LIN {X 0,Y 488.763,Z 747.858,A -85,B 0,C 180,E1 22935.063,E2 22935.063} C_VEL
LIN {X 0,Y 489.433,Z 736.714,A -85,B 0,C 180,E1 22932.524,E2 22932.524} C_VEL
LIN {X 0,Y 490.367,Z 723.912,A -85,B 0,C 180,E1 22930.092,E2 22930.092} C_VEL
LIN {X 0,Y 491.563,Z 709.449,A -85,B 0,C 180,E1 22927.769,E2 22927.769} C_VEL
LIN {X 0,Y 493.023,Z 693.233,A -85,B 0,C 180,E1 22925.561,E2 22925.561} C_VEL
LIN {X 0,Y 494.639,Z 676.036,A -85,B 0,C 180,E1 22923.569,E2 22923.569} C_VEL
LIN {X 0,Y 496.38,Z 657.448,A -85,B 0,C 180,E1 22921.747,E2 22921.747} C_VEL
LIN {X 0,Y 498.101,Z 638.983,A -85,B 0,C 180,E1 22920.21,E2 22920.21} C_VEL
LIN {X 0,Y 499.849,Z 618.816,A -85,B 0,C 180,E1 22918.796,E2 22918.796} C_VEL
LIN {X 0,Y 501.367,Z 599.666,A -85,B 0,C 180,E1 22917.692,E2 22917.692} C_VEL
LIN {X 0,Y 502.665,Z 578.619,A -85,B 0,C 180,E1 22916.736,E2 22916.736} C_VEL
LIN {X 0,Y 503.879,Z 555.736,A -85,B 0,C 180,E1 22915.926,E2 22915.926} C_VEL
LIN {X 0,Y 504.882,Z 532.422,A -85,B 0,C 180,E1 22915.329,E2 22915.329} C_VEL
LIN {X 0,Y 505.632,Z 495.194,A -85,B 0,C 180,E1 22914.703,E2 22914.703} C_VEL
LIN {X 0,Y 506.044,Z 485.944,A -85,B 0,C 180,E1 22914.556,E2 22914.556} C_VEL
LIN {X 0,Y 510.084,Z 468.745,A -85,B 0,C 180,E1 22913.911,E2 22913.911} C_VEL
LIN {X 0,Y 515.233,Z 449.255,A -85,B 0,C 180,E1 22913.225,E2 22913.225} C_VEL
LIN {X 0,Y 520.98,Z 432.729,A -85,B 0,C 180,E1 22912.735,E2 22912.735} C_VEL
LIN {X 0,Y 525.125,Z 418.193,A -85,B 0,C 180,E1 22912.255,E2 22912.255} C_VEL
LIN {X 0,Y 532.74,Z 398.375,A -85,B 0,C 180,E1 22911.731,E2 22911.731} C_VEL
LIN {X 0,Y 544.808,Z 371.898,A -85,B 0,C 180,E1 22911.19,E2 22911.19} C_VEL
LIN {X 0,Y 552.914,Z 353.703,A -85,B 0,C 180,E1 22910.934,E2 22910.934} C_VEL
LIN {X 0,Y 556.995,Z 340.142,A -85,B 0,C 180,E1 22910.569,E2 22910.569} C_VEL
LIN {X 0,Y 565.45,Z 316.224,A -85,B 0,C 180,E1 22910.17,E2 22910.17} C_VEL
LIN {X 0,Y 574.832,Z 288.327,A -85,B 0,C 180,E1 22909.898,E2 22909.898} C_VEL
LIN {X 0,Y 577.335,Z 280.017,A -85,B 0,C 180,E1 22909.834,E2 22909.834} C_VEL
LIN {X 0,Y 575.602,Z 280.443,A -85,B 0,C 180,E1 22909.221,E2 22909.221} C_VEL
LIN {X 0,Y 572.536,Z 280.47,A -85,B 0,C 180,E1 22908.671,E2 22908.671} C_VEL
LIN {X 0,Y 567.829,Z 279.596,A -85,B 0,C 180,E1 22908.145,E2 22908.145} C_VEL
LIN {X 0,Y 556.51,Z 275.352,A -85,B 0,C 180,E1 22907.141,E2 22907.141} C_VEL
LIN {X 0,Y 546.549,Z 269.641,A -85,B 0,C 180,E1 22906.119,E2 22906.119} C_VEL
LIN {X 0,Y 532.658,Z 258.791,A -85,B 0,C 180,E1 22904.44,E2 22904.44} C_VEL
LIN {X 0,Y 524.421,Z 249.344,A -85,B 0,C 180,E1 22903.193,E2 22903.193} C_VEL
LIN {X 0,Y 518.357,Z 238.972,A -85,B 0,C 180,E1 22902.015,E2 22902.015} C_VEL
LIN {X 0,Y 507.707,Z 216,A -85,B 0,C 180,E1 22899.467,E2 22899.467} C_VEL
LIN {X 0,Y 499.256,Z 199.711,A -85,B 0,C 180,E1 22897.359,E2 22897.359} C_VEL
LIN {X 0,Y 493.765,Z 190.209,A -85,B 0,C 180,E1 22895.961,E2 22895.961} C_VEL
LIN {X 0,Y 491.774,Z 186.487,A -85,B 0,C 180,E1 22895.412,E2 22895.412} C_VEL
LIN {X 0,Y 489.247,Z 182.669,A -85,B 0,C 180,E1 22894.759,E2 22894.759} C_VEL
LIN {X 0,Y 488.789,Z 180.844,A -85,B 0,C 180,E1 22894.515,E2 22894.515} C_VEL
LIN {X 0,Y 488.82,Z 181.07,A -85,B 0,C 180,E1 22894.37,E2 22894.37} C_VEL
LIN {X 0,Y 493.804,Z 196.293,A -85,B 0,C 180,E1 22893.002,E2 22893.002} C_VEL
LIN {X 0,Y 494.732,Z 233.032,A -85,B 0,C 180,E1 22890.281,E2 22890.281} C_VEL
LIN {X 0,Y 495.182,Z 268.429,A -85,B 0,C 180,E1 22887.476,E2 22887.476} C_VEL
LIN {X 0,Y 495.112,Z 303.332,A -85,B 0,C 180,E1 22884.582,E2 22884.582} C_VEL
LIN {X 0,Y 494.717,Z 328.2,A -85,B 0,C 180,E1 22882.456,E2 22882.456} C_VEL
LIN {X 0,Y 494.316,Z 330.636,A -85,B 0,C 180,E1 22882.319,E2 22882.319} C_VEL
LIN {X 0,Y 492.834,Z 451.64,A -85,B 0,C 180,E1 22880.353,E2 22880.353} C_VEL
LIN {X 0,Y 492.642,Z 497.502,A -85,B 0,C 180,E1 22879.623,E2 22879.623} C_VEL
LIN {X 0,Y 492.552,Z 514.82,A -85,B 0,C 180,E1 22879.126,E2 22879.126} C_VEL
LIN {X 0,Y 492.299,Z 531.833,A -85,B 0,C 180,E1 22878.41,E2 22878.41} C_VEL
LIN {X 0,Y 491.931,Z 547.816,A -85,B 0,C 180,E1 22877.506,E2 22877.506} C_VEL
LIN {X 0,Y 491.461,Z 562.541,A -85,B 0,C 180,E1 22876.426,E2 22876.426} C_VEL
LIN {X 0,Y 490.921,Z 576.831,A -85,B 0,C 180,E1 22875.111,E2 22875.111} C_VEL
LIN {X 0,Y 490.398,Z 589.354,A -85,B 0,C 180,E1 22873.68,E2 22873.68} C_VEL
LIN {X 0,Y 489.896,Z 600.231,A -85,B 0,C 180,E1 22872.135,E2 22872.135} C_VEL
LIN {X 0,Y 489.44,Z 610.273,A -85,B 0,C 180,E1 22870.356,E2 22870.356} C_VEL
LIN {X 0,Y 489.118,Z 618.168,A -85,B 0,C 180,E1 22868.582,E2 22868.582} C_VEL
LIN {X 0,Y 488.849,Z 624.536,A -85,B 0,C 180,E1 22866.695,E2 22866.695} C_VEL
LIN {X 0,Y 488.668,Z 629.357,A -85,B 0,C 180,E1 22864.694,E2 22864.694} C_VEL
LIN {X 0,Y 488.565,Z 632.392,A -85,B 0,C 180,E1 22862.698,E2 22862.698} C_VEL
LIN {X 0,Y 488.509,Z 633.701,A -85,B 0,C 180,E1 22860.703,E2 22860.703} C_VEL
LIN {X 0,Y 488.489,Z 633.33,A -85,B 0,C 180,E1 22858.709,E2 22858.709} C_VEL
LIN {X 0,Y 488.513,Z 631.151,A -85,B 0,C 180,E1 22856.597,E2 22856.597} C_VEL
LIN {X 0,Y 488.59,Z 627.335,A -85,B 0,C 180,E1 22854.598,E2 22854.598} C_VEL
LIN {X 0,Y 488.748,Z 621.608,A -85,B 0,C 180,E1 22852.595,E2 22852.595} C_VEL
LIN {X 0,Y 489.001,Z 614.344,A -85,B 0,C 180,E1 22850.704,E2 22850.704} C_VEL
LIN {X 0,Y 489.348,Z 605.609,A -85,B 0,C 180,E1 22848.926,E2 22848.926} C_VEL
LIN {X 0,Y 489.79,Z 595.341,A -85,B 0,C 180,E1 22847.263,E2 22847.263} C_VEL
LIN {X 0,Y 490.348,Z 583.074,A -85,B 0,C 180,E1 22845.655,E2 22845.655} C_VEL
LIN {X 0,Y 490.92,Z 570.214,A -85,B 0,C 180,E1 22844.283,E2 22844.283} C_VEL
LIN {X 0,Y 491.478,Z 556.401,A -85,B 0,C 180,E1 22843.087,E2 22843.087} C_VEL
LIN {X 0,Y 492.034,Z 540.803,A -85,B 0,C 180,E1 22842.008,E2 22842.008} C_VEL
LIN {X 0,Y 492.492,Z 524.476,A -85,B 0,C 180,E1 22841.129,E2 22841.129} C_VEL
LIN {X 0,Y 492.864,Z 507.517,A -85,B 0,C 180,E1 22840.456,E2 22840.456} C_VEL
LIN {X 0,Y 493.062,Z 489.747,A -85,B 0,C 180,E1 22839.985,E2 22839.985} C_VEL
LIN {X 0,Y 494.563,Z 326.51,A -85,B 0,C 180,E1 22837.4,E2 22837.4} C_VEL
LIN {X 0,Y 493.777,Z 321.369,A -85,B 0,C 180,E1 22837.246,E2 22837.246} C_VEL
LIN {X 0,Y 494.7,Z 284.617,A -85,B 0,C 180,E1 22833.817,E2 22833.817} C_VEL
LIN {X 0,Y 495.483,Z 247.552,A -85,B 0,C 180,E1 22830.369,E2 22830.369} C_VEL
LIN {X 0,Y 495.924,Z 219.277,A -85,B 0,C 180,E1 22827.745,E2 22827.745} C_VEL
LIN {X 0,Y 496.216,Z 218.46,A -85,B 0,C 180,E1 22827.507,E2 22827.507} C_VEL
LIN {X 0,Y 497.105,Z 219.551,A -85,B 0,C 180,E1 22827.105,E2 22827.105} C_VEL
LIN {X 0,Y 498.497,Z 223.242,A -85,B 0,C 180,E1 22826.646,E2 22826.646} C_VEL
LIN {X 0,Y 500.085,Z 229.6,A -85,B 0,C 180,E1 22826.249,E2 22826.249} C_VEL
LIN {X 0,Y 501.866,Z 239.61,A -85,B 0,C 180,E1 22825.842,E2 22825.842} C_VEL
LIN {X 0,Y 502.271,Z 247.308,A -85,B 0,C 180,E1 22825.659,E2 22825.659} C_VEL
LIN {X 0,Y 498.516,Z 445.436,A -85,B 0,C 180,E1 22822.414,E2 22822.414} C_VEL
LIN {X 0,Y 497.797,Z 472.996,A -85,B 0,C 180,E1 22821.899,E2 22821.899} C_VEL
LIN {X 0,Y 496.838,Z 494.838,A -85,B 0,C 180,E1 22821.269,E2 22821.269} C_VEL
LIN {X 0,Y 495.591,Z 515.448,A -85,B 0,C 180,E1 22820.462,E2 22820.462} C_VEL
LIN {X 0,Y 494.06,Z 535.344,A -85,B 0,C 180,E1 22819.458,E2 22819.458} C_VEL
LIN {X 0,Y 492.584,Z 552.464,A -85,B 0,C 180,E1 22818.413,E2 22818.413} C_VEL
LIN {X 0,Y 490.672,Z 572.409,A -85,B 0,C 180,E1 22816.949,E2 22816.949} C_VEL
LIN {X 0,Y 489.001,Z 588.827,A -85,B 0,C 180,E1 22815.529,E2 22815.529} C_VEL
LIN {X 0,Y 487.387,Z 604.827,A -85,B 0,C 180,E1 22813.939,E2 22813.939} C_VEL
LIN {X 0,Y 485.617,Z 622.035,A -85,B 0,C 180,E1 22811.938,E2 22811.938} C_VEL
LIN {X 0,Y 484.269,Z 635.641,A -85,B 0,C 180,E1 22810.104,E2 22810.104} C_VEL
LIN {X 0,Y 482.989,Z 649.658,A -85,B 0,C 180,E1 22807.933,E2 22807.933} C_VEL
LIN {X 0,Y 482.001,Z 661.364,A -85,B 0,C 180,E1 22805.797,E2 22805.797} C_VEL
LIN {X 0,Y 481.217,Z 672.009,A -85,B 0,C 180,E1 22803.552,E2 22803.552} C_VEL
LIN {X 0,Y 480.597,Z 682.358,A -85,B 0,C 180,E1 22800.922,E2 22800.922} C_VEL
LIN {X 0,Y 480.254,Z 689.801,A -85,B 0,C 180,E1 22798.61,E2 22798.61} C_VEL
LIN {X 0,Y 480.033,Z 696.665,A -85,B 0,C 180,E1 22795.939,E2 22795.939} C_VEL
LIN {X 0,Y 479.947,Z 701.157,A -85,B 0,C 180,E1 22793.559,E2 22793.559} C_VEL
LIN {X 0,Y 479.92,Z 704.361,A -85,B 0,C 180,E1 22791.127,E2 22791.127} C_VEL
LIN {X 0,Y 479.9,Z 706.187,A -85,B 0,C 180,E1 22788.463,E2 22788.463} C_VEL
LIN {X 0,Y 479.914,Z 706.33,A -85,B 0,C 180,E1 22786.087,E2 22786.087} C_VEL
LIN {X 0,Y 479.917,Z 705.127,A -85,B 0,C 180,E1 22783.617,E2 22783.617} C_VEL
LIN {X 0,Y 479.936,Z 702.064,A -85,B 0,C 180,E1 22780.929,E2 22780.929} C_VEL
LIN {X 0,Y 480,Z 697.765,A -85,B 0,C 180,E1 22778.505,E2 22778.505} C_VEL
LIN {X 0,Y 480.186,Z 691.783,A -85,B 0,C 180,E1 22775.976,E2 22775.976} C_VEL
LIN {X 0,Y 480.518,Z 683.988,A -85,B 0,C 180,E1 22773.46,E2 22773.46} C_VEL
LIN {X 0,Y 481.065,Z 674.571,A -85,B 0,C 180,E1 22770.953,E2 22770.953} C_VEL
LIN {X 0,Y 481.862,Z 663.093,A -85,B 0,C 180,E1 22768.454,E2 22768.454} C_VEL
LIN {X 0,Y 482.743,Z 652.276,A -85,B 0,C 180,E1 22766.438,E2 22766.438} C_VEL
LIN {X 0,Y 484.023,Z 638.341,A -85,B 0,C 180,E1 22764.191,E2 22764.191} C_VEL
LIN {X 0,Y 485.448,Z 623.716,A -85,B 0,C 180,E1 22762.187,E2 22762.187} C_VEL
LIN {X 0,Y 487.068,Z 608.002,A -85,B 0,C 180,E1 22760.309,E2 22760.309} C_VEL
LIN {X 0,Y 488.817,Z 590.709,A -85,B 0,C 180,E1 22758.556,E2 22758.556} C_VEL
LIN {X 0,Y 490.405,Z 574.812,A -85,B 0,C 180,E1 22757.16,E2 22757.16} C_VEL
LIN {X 0,Y 492.33,Z 555.785,A -85,B 0,C 180,E1 22755.715,E2 22755.715} C_VEL
LIN {X 0,Y 493.921,Z 537.357,A -85,B 0,C 180,E1 22754.562,E2 22754.562} C_VEL
LIN {X 0,Y 495.381,Z 518.625,A -85,B 0,C 180,E1 22753.586,E2 22753.586} C_VEL
LIN {X 0,Y 496.824,Z 496.661,A -85,B 0,C 180,E1 22752.691,E2 22752.691} C_VEL
LIN {X 0,Y 497.85,Z 474.503,A -85,B 0,C 180,E1 22752.025,E2 22752.025} C_VEL
LIN {X 0,Y 498.582,Z 449.883,A -85,B 0,C 180,E1 22751.541,E2 22751.541} C_VEL
LIN {X 0,Y 502.344,Z 259.982,A -85,B 0,C 180,E1 22748.409,E2 22748.409} C_VEL
LIN {X 0,Y 503.199,Z 216.754,A -85,B 0,C 180,E1 22747.677,E2 22747.677} C_VEL
LIN {X 0,Y 492.328,Z 199.865,A -85,B 0,C 180,E1 22746.266,E2 22746.266} C_VEL
LIN {X 0,Y 486.193,Z 190.932,A -85,B 0,C 180,E1 22745.443,E2 22745.443} C_VEL
LIN {X 0,Y 483.497,Z 186.812,A -85,B 0,C 180,E1 22745.069,E2 22745.069} C_VEL
LIN {X 0,Y 481.403,Z 183.82,A -85,B 0,C 180,E1 22744.779,E2 22744.779} C_VEL
LIN {X 0,Y 480.893,Z 181.877,A -85,B 0,C 180,E1 22744.631,E2 22744.631} C_VEL
LIN {X 0,Y 480.883,Z 181.825,A -85,B 0,C 180,E1 22741.023,E2 22741.023} C_VEL
LIN {X 0,Y 480.846,Z 181.833,A -85,B 0,C 180,E1 22737.556,E2 22737.556} C_VEL
LIN {X 0,Y 480.828,Z 181.84,A -85,B 0,C 180,E1 22733.951,E2 22733.951} C_VEL
LIN {X 0,Y 480.866,Z 181.837,A -85,B 0,C 180,E1 22730.482,E2 22730.482} C_VEL
LIN {X 0,Y 480.892,Z 181.835,A -85,B 0,C 180,E1 22727.002,E2 22727.002} C_VEL
LIN {X 0,Y 480.881,Z 181.834,A -85,B 0,C 180,E1 22723.326,E2 22723.326} C_VEL
LIN {X 0,Y 480.865,Z 181.831,A -85,B 0,C 180,E1 22719.669,E2 22719.669} C_VEL
LIN {X 0,Y 480.862,Z 181.825,A -85,B 0,C 180,E1 22716.195,E2 22716.195} C_VEL
LIN {X 0,Y 480.873,Z 181.823,A -85,B 0,C 180,E1 22712.584,E2 22712.584} C_VEL
LIN {X 0,Y 480.896,Z 181.83,A -85,B 0,C 180,E1 22708.977,E2 22708.977} C_VEL
LIN {X 0,Y 480.889,Z 181.836,A -85,B 0,C 180,E1 22705.361,E2 22705.361} C_VEL
LIN {X 0,Y 480.89,Z 181.825,A -85,B 0,C 180,E1 22701.722,E2 22701.722} C_VEL
LIN {X 0,Y 480.889,Z 181.821,A -85,B 0,C 180,E1 22698.16,E2 22698.16} C_VEL
LIN {X 0,Y 480.888,Z 181.828,A -85,B 0,C 180,E1 22694.572,E2 22694.572} C_VEL
LIN {X 0,Y 480.871,Z 181.839,A -85,B 0,C 180,E1 22690.907,E2 22690.907} C_VEL
LIN {X 0,Y 480.871,Z 181.831,A -85,B 0,C 180,E1 22687.338,E2 22687.338} C_VEL
LIN {X 0,Y 480.88,Z 181.822,A -85,B 0,C 180,E1 22683.696,E2 22683.696} C_VEL
LIN {X 0,Y 480.89,Z 181.823,A -85,B 0,C 180,E1 22680.12,E2 22680.12} C_VEL
LIN {X 0,Y 480.882,Z 181.829,A -85,B 0,C 180,E1 22676.544,E2 22676.544} C_VEL
LIN {X 0,Y 480.834,Z 181.84,A -85,B 0,C 180,E1 22673.073,E2 22673.073} C_VEL
LIN {X 0,Y 480.843,Z 181.839,A -85,B 0,C 180,E1 22669.457,E2 22669.457} C_VEL
LIN {X 0,Y 480.865,Z 181.836,A -85,B 0,C 180,E1 22665.797,E2 22665.797} C_VEL
LIN {X 0,Y 480.887,Z 181.829,A -85,B 0,C 180,E1 22662.204,E2 22662.204} C_VEL
LIN {X 0,Y 480.875,Z 181.824,A -85,B 0,C 180,E1 22658.662,E2 22658.662} C_VEL
LIN {X 0,Y 480.844,Z 181.835,A -85,B 0,C 180,E1 22655.164,E2 22655.164} C_VEL
LIN {X 0,Y 480.863,Z 181.881,A -85,B 0,C 180,E1 22653.845,E2 22653.845} C_VEL
LIN {X 0,Y 481.911,Z 184.96,A -85,B 0,C 180,E1 22653.375,E2 22653.375} C_VEL
LIN {X 0,Y 483.361,Z 187.323,A -85,B 0,C 180,E1 22652.93,E2 22652.93} C_VEL
LIN {X 0,Y 490.426,Z 201.495,A -85,B 0,C 180,E1 22650.572,E2 22650.572} C_VEL
LIN {X 0,Y 498.189,Z 217.501,A -85,B 0,C 180,E1 22648.098,E2 22648.098} C_VEL
LIN {X 0,Y 504.131,Z 230.513,A -85,B 0,C 180,E1 22646.236,E2 22646.236} C_VEL
LIN {X 0,Y 501.407,Z 270.851,A -85,B 0,C 180,E1 22642.971,E2 22642.971} C_VEL
LIN {X 0,Y 500.283,Z 297.085,A -85,B 0,C 180,E1 22640.836,E2 22640.836} C_VEL
LIN {X 0,Y 501.428,Z 313.16,A -85,B 0,C 180,E1 22639.38,E2 22639.38} C_VEL
LIN {X 0,Y 504.425,Z 327.463,A -85,B 0,C 180,E1 22637.935,E2 22637.935} C_VEL
LIN {X 0,Y 508.961,Z 339.677,A -85,B 0,C 180,E1 22636.562,E2 22636.562} C_VEL
LIN {X 0,Y 514.631,Z 349.651,A -85,B 0,C 180,E1 22635.307,E2 22635.307} C_VEL
LIN {X 0,Y 522.401,Z 359.052,A -85,B 0,C 180,E1 22633.975,E2 22633.975} C_VEL
LIN {X 0,Y 531.862,Z 366.96,A -85,B 0,C 180,E1 22632.689,E2 22632.689} C_VEL
LIN {X 0,Y 542.304,Z 372.999,A -85,B 0,C 180,E1 22631.535,E2 22631.535} C_VEL
LIN {X 0,Y 553.572,Z 377.39,A -85,B 0,C 180,E1 22630.5,E2 22630.5} C_VEL
LIN {X 0,Y 558.618,Z 378.484,A -85,B 0,C 180,E1 22629.998,E2 22629.998} C_VEL
LIN {X 0,Y 562.474,Z 378.433,A -85,B 0,C 180,E1 22629.407,E2 22629.407} C_VEL
LIN {X 0,Y 552.722,Z 394.402,A -85,B 0,C 180,E1 22629.264,E2 22629.264} C_VEL
LIN {X 0,Y 541.309,Z 410.43,A -85,B 0,C 180,E1 22628.956,E2 22628.956} C_VEL
LIN {X 0,Y 529.416,Z 427.314,A -85,B 0,C 180,E1 22628.484,E2 22628.484} C_VEL
LIN {X 0,Y 521.905,Z 440.164,A -85,B 0,C 180,E1 22628.019,E2 22628.019} C_VEL
LIN {X 0,Y 517.755,Z 448.383,A -85,B 0,C 180,E1 22627.677,E2 22627.677} C_VEL
LIN {X 0,Y 510.28,Z 461.224,A -85,B 0,C 180,E1 22627.192,E2 22627.192} C_VEL
LIN {X 0,Y 505.2,Z 472.975,A -85,B 0,C 180,E1 22626.634,E2 22626.634} C_VEL
LIN {X 0,Y 500.378,Z 484.799,A -85,B 0,C 180,E1 22626.049,E2 22626.049} C_VEL
LIN {X 0,Y 499.755,Z 487.325,A -85,B 0,C 180,E1 22625.95,E2 22625.95} C_VEL
LIN {X 0,Y 499.165,Z 500.84,A -85,B 0,C 180,E1 22625.764,E2 22625.764} C_VEL
LIN {X 0,Y 498.362,Z 532.024,A -85,B 0,C 180,E1 22625.213,E2 22625.213} C_VEL
LIN {X 0,Y 497.262,Z 554.109,A -85,B 0,C 180,E1 22624.63,E2 22624.63} C_VEL
LIN {X 0,Y 495.862,Z 576.831,A -85,B 0,C 180,E1 22623.816,E2 22623.816} C_VEL
LIN {X 0,Y 494.367,Z 598.257,A -85,B 0,C 180,E1 22622.822,E2 22622.822} C_VEL
LIN {X 0,Y 492.71,Z 618.983,A -85,B 0,C 180,E1 22621.64,E2 22621.64} C_VEL
LIN {X 0,Y 491.015,Z 638.957,A -85,B 0,C 180,E1 22620.264,E2 22620.264} C_VEL
LIN {X 0,Y 489.156,Z 657.45,A -85,B 0,C 180,E1 22618.708,E2 22618.708} C_VEL
LIN {X 0,Y 487.259,Z 676.275,A -85,B 0,C 180,E1 22616.836,E2 22616.836} C_VEL
LIN {X 0,Y 485.426,Z 694.22,A -85,B 0,C 180,E1 22614.716,E2 22614.716} C_VEL
LIN {X 0,Y 483.856,Z 710.291,A -85,B 0,C 180,E1 22612.476,E2 22612.476} C_VEL
LIN {X 0,Y 482.563,Z 724.626,A -85,B 0,C 180,E1 22610.117,E2 22610.117} C_VEL
LIN {X 0,Y 481.548,Z 737.378,A -85,B 0,C 180,E1 22607.629,E2 22607.629} C_VEL
LIN {X 0,Y 480.829,Z 748.339,A -85,B 0,C 180,E1 22605.066,E2 22605.066} C_VEL
LIN {X 0,Y 480.345,Z 757.699,A -85,B 0,C 180,E1 22602.38,E2 22602.38} C_VEL
LIN {X 0,Y 480.073,Z 765.002,A -85,B 0,C 180,E1 22599.712,E2 22599.712} C_VEL
LIN {X 0,Y 479.969,Z 770.228,A -85,B 0,C 180,E1 22597.18,E2 22597.18} C_VEL
LIN {X 0,Y 479.923,Z 773.872,A -85,B 0,C 180,E1 22594.66,E2 22594.66} C_VEL
LIN {X 0,Y 479.91,Z 775.982,A -85,B 0,C 180,E1 22592.03,E2 22592.03} C_VEL
LIN {X 0,Y 479.899,Z 776.434,A -85,B 0,C 180,E1 22589.403,E2 22589.403} C_VEL
LIN {X 0,Y 479.915,Z 775.326,A -85,B 0,C 180,E1 22586.895,E2 22586.895} C_VEL
LIN {X 0,Y 479.934,Z 772.505,A -85,B 0,C 180,E1 22584.261,E2 22584.261} C_VEL
LIN {X 0,Y 480.007,Z 767.958,A -85,B 0,C 180,E1 22581.616,E2 22581.616} C_VEL
LIN {X 0,Y 480.173,Z 761.915,A -85,B 0,C 180,E1 22579.077,E2 22579.077} C_VEL
LIN {X 0,Y 480.512,Z 754.11,A -85,B 0,C 180,E1 22576.523,E2 22576.523} C_VEL
LIN {X 0,Y 481.07,Z 744.373,A -85,B 0,C 180,E1 22573.953,E2 22573.953} C_VEL
LIN {X 0,Y 481.88,Z 733.088,A -85,B 0,C 180,E1 22571.483,E2 22571.483} C_VEL
LIN {X 0,Y 483.004,Z 719.562,A -85,B 0,C 180,E1 22569.004,E2 22569.004} C_VEL
LIN {X 0,Y 484.422,Z 704.354,A -85,B 0,C 180,E1 22566.653,E2 22566.653} C_VEL
LIN {X 0,Y 486.078,Z 687.709,A -85,B 0,C 180,E1 22564.472,E2 22564.472} C_VEL
LIN {X 0,Y 487.916,Z 669.751,A -85,B 0,C 180,E1 22562.477,E2 22562.477} C_VEL
LIN {X 0,Y 489.814,Z 651.146,A -85,B 0,C 180,E1 22560.732,E2 22560.732} C_VEL
LIN {X 0,Y 491.449,Z 633.867,A -85,B 0,C 180,E1 22559.36,E2 22559.36} C_VEL
LIN {X 0,Y 493.178,Z 612.483,A -85,B 0,C 180,E1 22557.983,E2 22557.983} C_VEL
LIN {X 0,Y 494.828,Z 590.016,A -85,B 0,C 180,E1 22556.798,E2 22556.798} C_VEL
LIN {X 0,Y 496.33,Z 566.99,A -85,B 0,C 180,E1 22555.84,E2 22555.84} C_VEL
LIN {X 0,Y 497.6,Z 543.342,A -85,B 0,C 180,E1 22555.098,E2 22555.098} C_VEL
LIN {X 0,Y 498.579,Z 519.122,A -85,B 0,C 180,E1 22554.578,E2 22554.578} C_VEL
LIN {X 0,Y 499.409,Z 484.886,A -85,B 0,C 180,E1 22554.047,E2 22554.047} C_VEL
LIN {X 0,Y 499.826,Z 481.764,A -85,B 0,C 180,E1 22553.976,E2 22553.976} C_VEL
LIN {X 0,Y 503.457,Z 467.078,A -85,B 0,C 180,E1 22553.43,E2 22553.43} C_VEL
LIN {X 0,Y 508.286,Z 448.826,A -85,B 0,C 180,E1 22552.779,E2 22552.779} C_VEL
LIN {X 0,Y 514.08,Z 432.325,A -85,B 0,C 180,E1 22552.288,E2 22552.288} C_VEL
LIN {X 0,Y 518.236,Z 417.779,A -85,B 0,C 180,E1 22551.803,E2 22551.803} C_VEL
LIN {X 0,Y 525.82,Z 397.929,A -85,B 0,C 180,E1 22551.273,E2 22551.273} C_VEL
LIN {X 0,Y 537.765,Z 371.828,A -85,B 0,C 180,E1 22550.721,E2 22550.721} C_VEL
LIN {X 0,Y 547.044,Z 352.733,A -85,B 0,C 180,E1 22550.365,E2 22550.365} C_VEL
LIN {X 0,Y 551.759,Z 338.349,A -85,B 0,C 180,E1 22549.961,E2 22549.961} C_VEL
LIN {X 0,Y 561.633,Z 313.909,A -85,B 0,C 180,E1 22549.473,E2 22549.473} C_VEL
LIN {X 0,Y 572.046,Z 287.955,A -85,B 0,C 180,E1 22549.131,E2 22549.131} C_VEL
LIN {X 0,Y 567.954,Z 287.614,A -85,B 0,C 180,E1 22548.586,E2 22548.586} C_VEL
LIN {X 0,Y 559.63,Z 285.196,A -85,B 0,C 180,E1 22547.855,E2 22547.855} C_VEL
LIN {X 0,Y 548.522,Z 280.226,A -85,B 0,C 180,E1 22546.813,E2 22546.813} C_VEL
LIN {X 0,Y 538.803,Z 273.883,A -85,B 0,C 180,E1 22545.75,E2 22545.75} C_VEL
LIN {X 0,Y 527.037,Z 264.39,A -85,B 0,C 180,E1 22544.278,E2 22544.278} C_VEL
LIN {X 0,Y 518.9,Z 254.887,A -85,B 0,C 180,E1 22543.009,E2 22543.009} C_VEL
LIN {X 0,Y 512.886,Z 244.581,A -85,B 0,C 180,E1 22541.814,E2 22541.814} C_VEL
LIN {X 0,Y 502.056,Z 220.958,A -85,B 0,C 180,E1 22539.147,E2 22539.147} C_VEL
LIN {X 0,Y 494.039,Z 205.355,A -85,B 0,C 180,E1 22537.092,E2 22537.092} C_VEL
LIN {X 0,Y 488.186,Z 195.267,A -85,B 0,C 180,E1 22535.567,E2 22535.567} C_VEL
LIN {X 0,Y 486.235,Z 191.59,A -85,B 0,C 180,E1 22535.009,E2 22535.009} C_VEL
LIN {X 0,Y 484.101,Z 188.655,A -85,B 0,C 180,E1 22534.466,E2 22534.466} C_VEL
LIN {X 0,Y 483.218,Z 188.203,A -85,B 0,C 180,E1 22534.286,E2 22534.286} C_VEL
LIN {X 0,Y 486.664,Z 199.47,A -85,B 0,C 180,E1 22533.26,E2 22533.26} C_VEL
LIN {X 0,Y 487.512,Z 236.04,A -85,B 0,C 180,E1 22530.526,E2 22530.526} C_VEL
LIN {X 0,Y 487.896,Z 270.354,A -85,B 0,C 180,E1 22527.789,E2 22527.789} C_VEL
LIN {X 0,Y 487.857,Z 303.401,A -85,B 0,C 180,E1 22525.058,E2 22525.058} C_VEL
LIN {X 0,Y 487.402,Z 329.74,A -85,B 0,C 180,E1 22522.812,E2 22522.812} C_VEL
LIN {X 0,Y 486.87,Z 332.626,A -85,B 0,C 180,E1 22522.637,E2 22522.637} C_VEL
LIN {X 0,Y 485.199,Z 453.648,A -85,B 0,C 180,E1 22520.611,E2 22520.611} C_VEL
LIN {X 0,Y 485.007,Z 499.094,A -85,B 0,C 180,E1 22519.87,E2 22519.87} C_VEL
LIN {X 0,Y 484.919,Z 516.446,A -85,B 0,C 180,E1 22519.364,E2 22519.364} C_VEL
LIN {X 0,Y 484.662,Z 533.219,A -85,B 0,C 180,E1 22518.648,E2 22518.648} C_VEL
LIN {X 0,Y 484.28,Z 549.271,A -85,B 0,C 180,E1 22517.73,E2 22517.73} C_VEL
LIN {X 0,Y 483.793,Z 564.065,A -85,B 0,C 180,E1 22516.633,E2 22516.633} C_VEL
LIN {X 0,Y 483.25,Z 577.809,A -85,B 0,C 180,E1 22515.357,E2 22515.357} C_VEL
LIN {X 0,Y 482.695,Z 590.465,A -85,B 0,C 180,E1 22513.903,E2 22513.903} C_VEL
LIN {X 0,Y 482.155,Z 601.433,A -85,B 0,C 180,E1 22512.333,E2 22512.333} C_VEL
LIN {X 0,Y 481.66,Z 611.533,A -85,B 0,C 180,E1 22510.525,E2 22510.525} C_VEL
LIN {X 0,Y 481.307,Z 619.483,A -85,B 0,C 180,E1 22508.722,E2 22508.722} C_VEL
LIN {X 0,Y 481.013,Z 625.894,A -85,B 0,C 180,E1 22506.804,E2 22506.804} C_VEL
LIN {X 0,Y 480.81,Z 630.73,A -85,B 0,C 180,E1 22504.771,E2 22504.771} C_VEL
LIN {X 0,Y 480.691,Z 633.761,A -85,B 0,C 180,E1 22502.742,E2 22502.742} C_VEL
LIN {X 0,Y 480.625,Z 635.054,A -85,B 0,C 180,E1 22500.715,E2 22500.715} C_VEL
LIN {X 0,Y 480.6,Z 634.648,A -85,B 0,C 180,E1 22498.688,E2 22498.688} C_VEL
LIN {X 0,Y 480.626,Z 632.429,A -85,B 0,C 180,E1 22496.541,E2 22496.541} C_VEL
LIN {X 0,Y 480.712,Z 628.55,A -85,B 0,C 180,E1 22494.509,E2 22494.509} C_VEL
LIN {X 0,Y 480.885,Z 622.75,A -85,B 0,C 180,E1 22492.473,E2 22492.473} C_VEL
LIN {X 0,Y 481.161,Z 615.416,A -85,B 0,C 180,E1 22490.551,E2 22490.551} C_VEL
LIN {X 0,Y 481.536,Z 606.578,A -85,B 0,C 180,E1 22488.744,E2 22488.744} C_VEL
LIN {X 0,Y 482.012,Z 596.194,A -85,B 0,C 180,E1 22487.054,E2 22487.054} C_VEL
LIN {X 0,Y 482.61,Z 583.809,A -85,B 0,C 180,E1 22485.42,E2 22485.42} C_VEL
LIN {X 0,Y 483.217,Z 570.791,A -85,B 0,C 180,E1 22484.026,E2 22484.026} C_VEL
LIN {X 0,Y 483.832,Z 555.974,A -85,B 0,C 180,E1 22482.749,E2 22482.749} C_VEL
LIN {X 0,Y 484.429,Z 539.968,A -85,B 0,C 180,E1 22481.653,E2 22481.653} C_VEL
LIN {X 0,Y 484.886,Z 524.04,A -85,B 0,C 180,E1 22480.808,E2 22480.808} C_VEL
LIN {X 0,Y 485.252,Z 506.64,A -85,B 0,C 180,E1 22480.136,E2 22480.136} C_VEL
LIN {X 0,Y 485.445,Z 488.575,A -85,B 0,C 180,E1 22479.673,E2 22479.673} C_VEL
LIN {X 0,Y 487.101,Z 327.578,A -85,B 0,C 180,E1 22477.076,E2 22477.076} C_VEL
LIN {X 0,Y 486.307,Z 322.646,A -85,B 0,C 180,E1 22476.941,E2 22476.941} C_VEL
LIN {X 0,Y 487.266,Z 285.092,A -85,B 0,C 180,E1 22473.427,E2 22473.427} C_VEL
LIN {X 0,Y 488.115,Z 247.825,A -85,B 0,C 180,E1 22469.944,E2 22469.944} C_VEL
LIN {X 0,Y 488.589,Z 221.292,A -85,B 0,C 180,E1 22467.457,E2 22467.457} C_VEL
LIN {X 0,Y 490.1,Z 222.979,A -85,B 0,C 180,E1 22467.273,E2 22467.273} C_VEL
LIN {X 0,Y 492.467,Z 223.168,A -85,B 0,C 180,E1 22467.035,E2 22467.035} C_VEL
LIN {X 0,Y 495.879,Z 221.24,A -85,B 0,C 180,E1 22466.739,E2 22466.739} C_VEL
LIN {X 0,Y 496.774,Z 220.421,A -85,B 0,C 180,E1 22466.669,E2 22466.669} C_VEL
LIN {X 0,Y 500.842,Z 220.212,A -85,B 0,C 180,E1 22466.29,E2 22466.29} C_VEL
LIN {X 0,Y 502.856,Z 219.573,A -85,B 0,C 180,E1 22466.115,E2 22466.115} C_VEL
LIN {X 0,Y 502.271,Z 247.308,A -85,B 0,C 180,E1 22465.659,E2 22465.659} C_VEL
LIN {X 0,Y 501.337,Z 254.999,A -85,B 0,C 180,E1 22465.602,E2 22465.602} C_VEL
LIN {X 0,Y 495.997,Z 275.543,A -85,B 0,C 180,E1 22465.705,E2 22465.705} C_VEL
LIN {X 0,Y 495.24,Z 282.145,A -85,B 0,C 180,E1 22465.649,E2 22465.649} C_VEL
LIN {X 0,Y 491.275,Z 469.293,A -85,B 0,C 180,E1 22462.497,E2 22462.497} C_VEL
LIN {X 0,Y 490.314,Z 490.789,A -85,B 0,C 180,E1 22461.919,E2 22461.919} C_VEL
LIN {X 0,Y 489.071,Z 512.091,A -85,B 0,C 180,E1 22461.124,E2 22461.124} C_VEL
LIN {X 0,Y 487.528,Z 532.593,A -85,B 0,C 180,E1 22460.134,E2 22460.134} C_VEL
LIN {X 0,Y 485.821,Z 551.405,A -85,B 0,C 180,E1 22459.001,E2 22459.001} C_VEL
LIN {X 0,Y 483.931,Z 570.524,A -85,B 0,C 180,E1 22457.616,E2 22457.616} C_VEL
LIN {X 0,Y 481.913,Z 588.476,A -85,B 0,C 180,E1 22456.05,E2 22456.05} C_VEL
LIN {X 0,Y 480.141,Z 604.065,A -85,B 0,C 180,E1 22454.465,E2 22454.465} C_VEL
LIN {X 0,Y 478.212,Z 621.436,A -85,B 0,C 180,E1 22452.433,E2 22452.433} C_VEL
LIN {X 0,Y 476.738,Z 635.221,A -85,B 0,C 180,E1 22450.554,E2 22450.554} C_VEL
LIN {X 0,Y 475.315,Z 649.522,A -85,B 0,C 180,E1 22448.313,E2 22448.313} C_VEL
LIN {X 0,Y 474.176,Z 661.764,A -85,B 0,C 180,E1 22446.037,E2 22446.037} C_VEL
LIN {X 0,Y 473.303,Z 672.781,A -85,B 0,C 180,E1 22443.66,E2 22443.66} C_VEL
LIN {X 0,Y 472.647,Z 682.75,A -85,B 0,C 180,E1 22441.045,E2 22441.045} C_VEL
LIN {X 0,Y 472.282,Z 690.05,A -85,B 0,C 180,E1 22438.723,E2 22438.723} C_VEL
LIN {X 0,Y 472.044,Z 696.845,A -85,B 0,C 180,E1 22436.006,E2 22436.006} C_VEL
LIN {X 0,Y 471.95,Z 701.258,A -85,B 0,C 180,E1 22433.604,E2 22433.604} C_VEL
LIN {X 0,Y 471.92,Z 704.451,A -85,B 0,C 180,E1 22431.111,E2 22431.111} C_VEL
LIN {X 0,Y 471.902,Z 706.218,A -85,B 0,C 180,E1 22428.337,E2 22428.337} C_VEL
LIN {X 0,Y 471.914,Z 706.31,A -85,B 0,C 180,E1 22425.988,E2 22425.988} C_VEL
LIN {X 0,Y 471.914,Z 705.062,A -85,B 0,C 180,E1 22423.466,E2 22423.466} C_VEL
LIN {X 0,Y 471.935,Z 701.936,A -85,B 0,C 180,E1 22420.745,E2 22420.745} C_VEL
LIN {X 0,Y 472.008,Z 697.849,A -85,B 0,C 180,E1 22418.405,E2 22418.405} C_VEL
LIN {X 0,Y 472.214,Z 691.903,A -85,B 0,C 180,E1 22415.834,E2 22415.834} C_VEL
LIN {X 0,Y 472.578,Z 684.141,A -85,B 0,C 180,E1 22413.275,E2 22413.275} C_VEL
LIN {X 0,Y 473.098,Z 675.695,A -85,B 0,C 180,E1 22410.969,E2 22410.969} C_VEL
LIN {X 0,Y 473.994,Z 663.93,A -85,B 0,C 180,E1 22408.308,E2 22408.308} C_VEL
LIN {X 0,Y 474.935,Z 653.215,A -85,B 0,C 180,E1 22406.258,E2 22406.258} C_VEL
LIN {X 0,Y 476.232,Z 640.251,A -85,B 0,C 180,E1 22404.095,E2 22404.095} C_VEL
LIN {X 0,Y 477.828,Z 624.999,A -85,B 0,C 180,E1 22401.941,E2 22401.941} C_VEL
LIN {X 0,Y 479.361,Z 610.953,A -85,B 0,C 180,E1 22400.213,E2 22400.213} C_VEL
LIN {X 0,Y 481.524,Z 592.016,A -85,B 0,C 180,E1 22398.198,E2 22398.198} C_VEL
LIN {X 0,Y 483.337,Z 575.769,A -85,B 0,C 180,E1 22396.725,E2 22396.725} C_VEL
LIN {X 0,Y 485.372,Z 556.761,A -85,B 0,C 180,E1 22395.262,E2 22395.262} C_VEL
LIN {X 0,Y 487.142,Z 537.344,A -85,B 0,C 180,E1 22394.036,E2 22394.036} C_VEL
LIN {X 0,Y 488.804,Z 517.208,A -85,B 0,C 180,E1 22392.992,E2 22392.992} C_VEL
LIN {X 0,Y 490.208,Z 495.852,A -85,B 0,C 180,E1 22392.135,E2 22392.135} C_VEL
LIN {X 0,Y 491.251,Z 473.547,A -85,B 0,C 180,E1 22391.48,E2 22391.48} C_VEL
LIN {X 0,Y 492.052,Z 445.081,A -85,B 0,C 180,E1 22390.941,E2 22390.941} C_VEL
LIN {X 0,Y 496.64,Z 240.16,A -85,B 0,C 180,E1 22387.486,E2 22387.486} C_VEL
LIN {X 0,Y 496.999,Z 220.048,A -85,B 0,C 180,E1 22387.133,E2 22387.133} C_VEL
LIN {X 0,Y 485.248,Z 201.887,A -85,B 0,C 180,E1 22385.562,E2 22385.562} C_VEL
LIN {X 0,Y 478.39,Z 192.058,A -85,B 0,C 180,E1 22384.616,E2 22384.616} C_VEL
LIN {X 0,Y 475.702,Z 187.924,A -85,B 0,C 180,E1 22384.23,E2 22384.23} C_VEL
LIN {X 0,Y 473.837,Z 185.604,A -85,B 0,C 180,E1 22383.966,E2 22383.966} C_VEL
LIN {X 0,Y 472.94,Z 182.815,A -85,B 0,C 180,E1 22383.47,E2 22383.47} C_VEL
LIN {X 0,Y 472.926,Z 182.826,A -85,B 0,C 180,E1 22379.85,E2 22379.85} C_VEL
LIN {X 0,Y 472.924,Z 182.825,A -85,B 0,C 180,E1 22376.364,E2 22376.364} C_VEL
LIN {X 0,Y 472.94,Z 182.818,A -85,B 0,C 180,E1 22372.797,E2 22372.797} C_VEL
LIN {X 0,Y 472.956,Z 182.814,A -85,B 0,C 180,E1 22369.187,E2 22369.187} C_VEL
LIN {X 0,Y 472.948,Z 182.816,A -85,B 0,C 180,E1 22365.592,E2 22365.592} C_VEL
LIN {X 0,Y 472.95,Z 182.818,A -85,B 0,C 180,E1 22361.913,E2 22361.913} C_VEL
LIN {X 0,Y 472.95,Z 182.823,A -85,B 0,C 180,E1 22358.275,E2 22358.275} C_VEL
LIN {X 0,Y 472.938,Z 182.823,A -85,B 0,C 180,E1 22354.66,E2 22354.66} C_VEL
LIN {X 0,Y 472.933,Z 182.814,A -85,B 0,C 180,E1 22351.055,E2 22351.055} C_VEL
LIN {X 0,Y 472.938,Z 182.81,A -85,B 0,C 180,E1 22347.445,E2 22347.445} C_VEL
LIN {X 0,Y 472.947,Z 182.815,A -85,B 0,C 180,E1 22343.816,E2 22343.816} C_VEL
LIN {X 0,Y 472.955,Z 182.824,A -85,B 0,C 180,E1 22340.157,E2 22340.157} C_VEL
LIN {X 0,Y 472.952,Z 182.819,A -85,B 0,C 180,E1 22336.457,E2 22336.457} C_VEL
LIN {X 0,Y 472.921,Z 182.812,A -85,B 0,C 180,E1 22332.827,E2 22332.827} C_VEL
LIN {X 0,Y 472.922,Z 182.815,A -85,B 0,C 180,E1 22329.247,E2 22329.247} C_VEL
LIN {X 0,Y 472.933,Z 182.825,A -85,B 0,C 180,E1 22325.703,E2 22325.703} C_VEL
LIN {X 0,Y 472.947,Z 182.823,A -85,B 0,C 180,E1 22322.06,E2 22322.06} C_VEL
LIN {X 0,Y 472.953,Z 182.819,A -85,B 0,C 180,E1 22318.426,E2 22318.426} C_VEL
LIN {X 0,Y 472.913,Z 182.819,A -85,B 0,C 180,E1 22314.906,E2 22314.906} C_VEL
LIN {X 0,Y 472.888,Z 182.819,A -85,B 0,C 180,E1 22311.367,E2 22311.367} C_VEL
LIN {X 0,Y 472.915,Z 182.817,A -85,B 0,C 180,E1 22307.671,E2 22307.671} C_VEL
LIN {X 0,Y 472.939,Z 182.819,A -85,B 0,C 180,E1 22304.048,E2 22304.048} C_VEL
LIN {X 0,Y 472.953,Z 182.822,A -85,B 0,C 180,E1 22300.359,E2 22300.359} C_VEL
LIN {X 0,Y 472.922,Z 182.825,A -85,B 0,C 180,E1 22296.844,E2 22296.844} C_VEL
LIN {X 0,Y 472.939,Z 183.012,A -85,B 0,C 180,E1 22294.881,E2 22294.881} C_VEL
LIN {X 0,Y 474.087,Z 186.056,A -85,B 0,C 180,E1 22294.384,E2 22294.384} C_VEL
LIN {X 0,Y 475.236,Z 187.613,A -85,B 0,C 180,E1 22294.049,E2 22294.049} C_VEL
LIN {X 0,Y 477.127,Z 191.604,A -85,B 0,C 180,E1 22293.356,E2 22293.356} C_VEL
LIN {X 0,Y 484.509,Z 206.345,A -85,B 0,C 180,E1 22290.855,E2 22290.855} C_VEL
LIN {X 0,Y 492.806,Z 223.596,A -85,B 0,C 180,E1 22288.163,E2 22288.163} C_VEL
LIN {X 0,Y 497.698,Z 234.386,A -85,B 0,C 180,E1 22286.602,E2 22286.602} C_VEL
LIN {X 0,Y 494.801,Z 274.277,A -85,B 0,C 180,E1 22283.343,E2 22283.343} C_VEL
LIN {X 0,Y 493.634,Z 299.777,A -85,B 0,C 180,E1 22281.244,E2 22281.244} C_VEL
LIN {X 0,Y 494.671,Z 315.781,A -85,B 0,C 180,E1 22279.783,E2 22279.783} C_VEL
LIN {X 0,Y 497.533,Z 330.338,A -85,B 0,C 180,E1 22278.304,E2 22278.304} C_VEL
LIN {X 0,Y 501.912,Z 342.825,A -85,B 0,C 180,E1 22276.899,E2 22276.899} C_VEL
LIN {X 0,Y 507.937,Z 353.894,A -85,B 0,C 180,E1 22275.511,E2 22275.511} C_VEL
LIN {X 0,Y 515.597,Z 363.517,A -85,B 0,C 180,E1 22274.151,E2 22274.151} C_VEL
LIN {X 0,Y 524.384,Z 371.334,A -85,B 0,C 180,E1 22272.899,E2 22272.899} C_VEL
LIN {X 0,Y 534.47,Z 377.751,A -85,B 0,C 180,E1 22271.719,E2 22271.719} C_VEL
LIN {X 0,Y 546.28,Z 382.926,A -85,B 0,C 180,E1 22270.574,E2 22270.574} C_VEL
LIN {X 0,Y 552.927,Z 385.067,A -85,B 0,C 180,E1 22269.997,E2 22269.997} C_VEL
LIN {X 0,Y 528.703,Z 417.299,A -85,B 0,C 180,E1 22269.241,E2 22269.241} C_VEL
LIN {X 0,Y 518.997,Z 432.295,A -85,B 0,C 180,E1 22268.764,E2 22268.764} C_VEL
LIN {X 0,Y 512.627,Z 444.592,A -85,B 0,C 180,E1 22268.263,E2 22268.263} C_VEL
LIN {X 0,Y 503.979,Z 459.365,A -85,B 0,C 180,E1 22267.709,E2 22267.709} C_VEL
LIN {X 0,Y 498.573,Z 471.599,A -85,B 0,C 180,E1 22267.131,E2 22267.131} C_VEL
LIN {X 0,Y 493.573,Z 484.129,A -85,B 0,C 180,E1 22266.528,E2 22266.528} C_VEL
LIN {X 0,Y 492.734,Z 497.7,A -85,B 0,C 180,E1 22266.359,E2 22266.359} C_VEL
LIN {X 0,Y 491.867,Z 529.417,A -85,B 0,C 180,E1 22265.796,E2 22265.796} C_VEL
LIN {X 0,Y 490.631,Z 552.073,A -85,B 0,C 180,E1 22265.199,E2 22265.199} C_VEL
LIN {X 0,Y 489.159,Z 573.938,A -85,B 0,C 180,E1 22264.414,E2 22264.414} C_VEL
LIN {X 0,Y 487.5,Z 595.718,A -85,B 0,C 180,E1 22263.41,E2 22263.41} C_VEL
LIN {X 0,Y 485.707,Z 616.675,A -85,B 0,C 180,E1 22262.214,E2 22262.214} C_VEL
LIN {X 0,Y 483.865,Z 636.828,A -85,B 0,C 180,E1 22260.828,E2 22260.828} C_VEL
LIN {X 0,Y 482.001,Z 656.048,A -85,B 0,C 180,E1 22259.264,E2 22259.264} C_VEL
LIN {X 0,Y 480.366,Z 672.142,A -85,B 0,C 180,E1 22257.723,E2 22257.723} C_VEL
LIN {X 0,Y 478.469,Z 689.295,A -85,B 0,C 180,E1 22255.756,E2 22255.756} C_VEL
LIN {X 0,Y 476.735,Z 705.457,A -85,B 0,C 180,E1 22253.578,E2 22253.578} C_VEL
LIN {X 0,Y 475.234,Z 720.352,A -85,B 0,C 180,E1 22251.215,E2 22251.215} C_VEL
LIN {X 0,Y 474.026,Z 733.739,A -85,B 0,C 180,E1 22248.7,E2 22248.7} C_VEL
LIN {X 0,Y 473.122,Z 745.412,A -85,B 0,C 180,E1 22246.072,E2 22246.072} C_VEL
LIN {X 0,Y 472.51,Z 755.348,A -85,B 0,C 180,E1 22243.335,E2 22243.335} C_VEL
LIN {X 0,Y 472.163,Z 763.204,A -85,B 0,C 180,E1 22240.616,E2 22240.616} C_VEL
LIN {X 0,Y 471.996,Z 769.154,A -85,B 0,C 180,E1 22237.914,E2 22237.914} C_VEL
LIN {X 0,Y 471.929,Z 773.226,A -85,B 0,C 180,E1 22235.274,E2 22235.274} C_VEL
LIN {X 0,Y 471.911,Z 775.642,A -85,B 0,C 180,E1 22232.671,E2 22232.671} C_VEL
LIN {X 0,Y 471.912,Z 776.5,A -85,B 0,C 180,E1 22230,E2 22230} C_VEL
LIN {X 0,Y 471.911,Z 775.642,A -85,B 0,C 180,E1 22227.328,E2 22227.328} C_VEL
LIN {X 0,Y 471.929,Z 773.225,A -85,B 0,C 180,E1 22224.726,E2 22224.726} C_VEL
LIN {X 0,Y 471.995,Z 769.153,A -85,B 0,C 180,E1 22222.085,E2 22222.085} C_VEL
LIN {X 0,Y 472.161,Z 763.204,A -85,B 0,C 180,E1 22219.383,E2 22219.383} C_VEL
LIN {X 0,Y 472.51,Z 755.347,A -85,B 0,C 180,E1 22216.664,E2 22216.664} C_VEL
LIN {X 0,Y 473.123,Z 745.411,A -85,B 0,C 180,E1 22213.928,E2 22213.928} C_VEL
LIN {X 0,Y 474.04,Z 733.594,A -85,B 0,C 180,E1 22211.269,E2 22211.269} C_VEL
LIN {X 0,Y 475.254,Z 720.145,A -85,B 0,C 180,E1 22208.748,E2 22208.748} C_VEL
LIN {X 0,Y 476.762,Z 705.217,A -85,B 0,C 180,E1 22206.386,E2 22206.386} C_VEL
LIN {X 0,Y 478.594,Z 688.227,A -85,B 0,C 180,E1 22204.11,E2 22204.11} C_VEL
LIN {X 0,Y 480.609,Z 669.976,A -85,B 0,C 180,E1 22202.047,E2 22202.047} C_VEL
LIN {X 0,Y 482.263,Z 653.381,A -85,B 0,C 180,E1 22200.508,E2 22200.508} C_VEL
LIN {X 0,Y 484.127,Z 632.973,A -85,B 0,C 180,E1 22198.914,E2 22198.914} C_VEL
LIN {X 0,Y 485.998,Z 611.427,A -85,B 0,C 180,E1 22197.512,E2 22197.512} C_VEL
LIN {X 0,Y 487.747,Z 589.455,A -85,B 0,C 180,E1 22196.333,E2 22196.333} C_VEL
LIN {X 0,Y 489.329,Z 567.194,A -85,B 0,C 180,E1 22195.386,E2 22195.386} C_VEL
LIN {X 0,Y 490.735,Z 543.919,A -85,B 0,C 180,E1 22194.627,E2 22194.627} C_VEL
LIN {X 0,Y 491.91,Z 519.829,A -85,B 0,C 180,E1 22194.073,E2 22194.073} C_VEL
LIN {X 0,Y 492.826,Z 485.119,A -85,B 0,C 180,E1 22193.522,E2 22193.522} C_VEL
LIN {X 0,Y 493.348,Z 478.804,A -85,B 0,C 180,E1 22193.427,E2 22193.427} C_VEL
LIN {X 0,Y 501.376,Z 448.356,A -85,B 0,C 180,E1 22192.321,E2 22192.321} C_VEL
LIN {X 0,Y 507.504,Z 430.662,A -85,B 0,C 180,E1 22191.784,E2 22191.784} C_VEL
LIN {X 0,Y 512.191,Z 414.991,A -85,B 0,C 180,E1 22191.269,E2 22191.269} C_VEL
LIN {X 0,Y 520.267,Z 394.355,A -85,B 0,C 180,E1 22190.73,E2 22190.73} C_VEL
LIN {X 0,Y 533.043,Z 366.858,A -85,B 0,C 180,E1 22190.165,E2 22190.165} C_VEL
LIN {X 0,Y 540.302,Z 352.322,A -85,B 0,C 180,E1 22189.909,E2 22189.909} C_VEL
LIN {X 0,Y 545.458,Z 336.797,A -85,B 0,C 180,E1 22189.472,E2 22189.472} C_VEL
LIN {X 0,Y 556.168,Z 311.444,A -85,B 0,C 180,E1 22188.922,E2 22188.922} C_VEL
LIN {X 0,Y 563.765,Z 294.649,A -85,B 0,C 180,E1 22188.608,E2 22188.608} C_VEL
LIN {X 0,Y 551.495,Z 290.5,A -85,B 0,C 180,E1 22187.552,E2 22187.552} C_VEL
LIN {X 0,Y 539.914,Z 284.439,A -85,B 0,C 180,E1 22186.393,E2 22186.393} C_VEL
LIN {X 0,Y 523.916,Z 272.348,A -85,B 0,C 180,E1 22184.458,E2 22184.458} C_VEL
LIN {X 0,Y 515.593,Z 263.368,A -85,B 0,C 180,E1 22183.2,E2 22183.2} C_VEL
LIN {X 0,Y 509.799,Z 254.713,A -85,B 0,C 180,E1 22182.125,E2 22182.125} C_VEL
LIN {X 0,Y 496.125,Z 225.336,A -85,B 0,C 180,E1 22178.745,E2 22178.745} C_VEL
LIN {X 0,Y 488.413,Z 210.296,A -85,B 0,C 180,E1 22176.71,E2 22176.71} C_VEL
LIN {X 0,Y 481.133,Z 197.361,A -85,B 0,C 180,E1 22174.709,E2 22174.709} C_VEL
LIN {X 0,Y 480.472,Z 196.549,A -85,B 0,C 180,E1 22174.546,E2 22174.546} C_VEL
LIN {X 0,Y 478.333,Z 196.442,A -85,B 0,C 180,E1 22174.214,E2 22174.214} C_VEL
LIN {X 0,Y 477.971,Z 196.329,A -85,B 0,C 180,E1 22174.114,E2 22174.114} C_VEL
LIN {X 0,Y 479.604,Z 202.756,A -85,B 0,C 180,E1 22173.536,E2 22173.536} C_VEL
LIN {X 0,Y 480.367,Z 239.025,A -85,B 0,C 180,E1 22170.799,E2 22170.799} C_VEL
LIN {X 0,Y 480.67,Z 270.035,A -85,B 0,C 180,E1 22168.312,E2 22168.312} C_VEL
LIN {X 0,Y 480.649,Z 301.566,A -85,B 0,C 180,E1 22165.711,E2 22165.711} C_VEL
LIN {X 0,Y 480.278,Z 330.454,A -85,B 0,C 180,E1 22163.235,E2 22163.235} C_VEL
LIN {X 0,Y 479.483,Z 334.49,A -85,B 0,C 180,E1 22162.979,E2 22162.979} C_VEL
LIN {X 0,Y 477.71,Z 446.329,A -85,B 0,C 180,E1 22161.038,E2 22161.038} C_VEL
LIN {X 0,Y 477.383,Z 500.238,A -85,B 0,C 180,E1 22160.137,E2 22160.137} C_VEL
LIN {X 0,Y 477.309,Z 517.569,A -85,B 0,C 180,E1 22159.632,E2 22159.632} C_VEL
LIN {X 0,Y 477.068,Z 533.465,A -85,B 0,C 180,E1 22158.956,E2 22158.956} C_VEL
LIN {X 0,Y 476.699,Z 548.871,A -85,B 0,C 180,E1 22158.084,E2 22158.084} C_VEL
LIN {X 0,Y 476.23,Z 563.456,A -85,B 0,C 180,E1 22157.03,E2 22157.03} C_VEL
LIN {X 0,Y 475.676,Z 577.028,A -85,B 0,C 180,E1 22155.795,E2 22155.795} C_VEL
LIN {X 0,Y 475.065,Z 590.098,A -85,B 0,C 180,E1 22154.317,E2 22154.317} C_VEL
LIN {X 0,Y 474.507,Z 601.119,A -85,B 0,C 180,E1 22152.782,E2 22152.782} C_VEL
LIN {X 0,Y 473.991,Z 611.013,A -85,B 0,C 180,E1 22151.067,E2 22151.067} C_VEL
LIN {X 0,Y 473.567,Z 619.351,A -85,B 0,C 180,E1 22149.233,E2 22149.233} C_VEL
LIN {X 0,Y 473.232,Z 626.189,A -85,B 0,C 180,E1 22147.283,E2 22147.283} C_VEL
LIN {X 0,Y 472.999,Z 631.167,A -85,B 0,C 180,E1 22145.336,E2 22145.336} C_VEL
LIN {X 0,Y 472.84,Z 634.569,A -85,B 0,C 180,E1 22143.273,E2 22143.273} C_VEL
LIN {X 0,Y 472.75,Z 636.293,A -85,B 0,C 180,E1 22141.09,E2 22141.09} C_VEL
LIN {X 0,Y 472.717,Z 636.198,A -85,B 0,C 180,E1 22139.03,E2 22139.03} C_VEL
LIN {X 0,Y 472.723,Z 634.374,A -85,B 0,C 180,E1 22136.969,E2 22136.969} C_VEL
LIN {X 0,Y 472.798,Z 630.834,A -85,B 0,C 180,E1 22134.904,E2 22134.904} C_VEL
LIN {X 0,Y 472.97,Z 625.468,A -85,B 0,C 180,E1 22132.835,E2 22132.835} C_VEL
LIN {X 0,Y 473.242,Z 618.52,A -85,B 0,C 180,E1 22130.882,E2 22130.882} C_VEL
LIN {X 0,Y 473.631,Z 609.464,A -85,B 0,C 180,E1 22128.924,E2 22128.924} C_VEL
LIN {X 0,Y 474.119,Z 599.497,A -85,B 0,C 180,E1 22127.206,E2 22127.206} C_VEL
LIN {X 0,Y 474.7,Z 588.048,A -85,B 0,C 180,E1 22125.608,E2 22125.608} C_VEL
LIN {X 0,Y 475.34,Z 575.014,A -85,B 0,C 180,E1 22124.13,E2 22124.13} C_VEL
LIN {X 0,Y 475.986,Z 560.983,A -85,B 0,C 180,E1 22122.834,E2 22122.834} C_VEL
LIN {X 0,Y 476.598,Z 546.013,A -85,B 0,C 180,E1 22121.721,E2 22121.721} C_VEL
LIN {X 0,Y 477.11,Z 529.95,A -85,B 0,C 180,E1 22120.79,E2 22120.79} C_VEL
LIN {X 0,Y 477.542,Z 512.391,A -85,B 0,C 180,E1 22120.029,E2 22120.029} C_VEL
LIN {X 0,Y 477.792,Z 494.881,A -85,B 0,C 180,E1 22119.507,E2 22119.507} C_VEL
LIN {X 0,Y 478.274,Z 442.265,A -85,B 0,C 180,E1 22118.628,E2 22118.628} C_VEL
LIN {X 0,Y 479.644,Z 328.584,A -85,B 0,C 180,E1 22116.74,E2 22116.74} C_VEL
LIN {X 0,Y 478.856,Z 323.567,A -85,B 0,C 180,E1 22116.593,E2 22116.593} C_VEL
LIN {X 0,Y 479.846,Z 285.83,A -85,B 0,C 180,E1 22113.05,E2 22113.05} C_VEL
LIN {X 0,Y 480.732,Z 249.533,A -85,B 0,C 180,E1 22109.641,E2 22109.641} C_VEL
LIN {X 0,Y 481.113,Z 232.424,A -85,B 0,C 180,E1 22108.015,E2 22108.015} C_VEL
LIN {X 0,Y 482.584,Z 234.009,A -85,B 0,C 180,E1 22107.827,E2 22107.827} C_VEL
LIN {X 0,Y 484.909,Z 234.105,A -85,B 0,C 180,E1 22107.58,E2 22107.58} C_VEL
LIN {X 0,Y 488.297,Z 232.123,A -85,B 0,C 180,E1 22107.276,E2 22107.276} C_VEL
LIN {X 0,Y 489.598,Z 231.137,A -85,B 0,C 180,E1 22107.166,E2 22107.166} C_VEL
LIN {X 0,Y 493.655,Z 230.773,A -85,B 0,C 180,E1 22106.773,E2 22106.773} C_VEL
LIN {X 0,Y 496.418,Z 229.647,A -85,B 0,C 180,E1 22106.53,E2 22106.53} C_VEL
LIN {X 0,Y 495.24,Z 282.145,A -85,B 0,C 180,E1 22105.649,E2 22105.649} C_VEL
LIN {X 0,Y 494.271,Z 289.835,A -85,B 0,C 180,E1 22105.593,E2 22105.593} C_VEL
LIN {X 0,Y 488.911,Z 310.372,A -85,B 0,C 180,E1 22105.689,E2 22105.689} C_VEL
LIN {X 0,Y 488.142,Z 316.969,A -85,B 0,C 180,E1 22105.631,E2 22105.631} C_VEL
LIN {X 0,Y 484.542,Z 471.093,A -85,B 0,C 180,E1 22102.982,E2 22102.982} C_VEL
LIN {X 0,Y 483.562,Z 492.341,A -85,B 0,C 180,E1 22102.399,E2 22102.399} C_VEL
LIN {X 0,Y 482.278,Z 513.414,A -85,B 0,C 180,E1 22101.598,E2 22101.598} C_VEL
LIN {X 0,Y 480.72,Z 533.375,A -85,B 0,C 180,E1 22100.626,E2 22100.626} C_VEL
LIN {X 0,Y 478.902,Z 552.5,A -85,B 0,C 180,E1 22099.462,E2 22099.462} C_VEL
LIN {X 0,Y 476.835,Z 572.052,A -85,B 0,C 180,E1 22098.017,E2 22098.017} C_VEL
LIN {X 0,Y 474.719,Z 589.952,A -85,B 0,C 180,E1 22096.431,E2 22096.431} C_VEL
LIN {X 0,Y 472.716,Z 606.495,A -85,B 0,C 180,E1 22094.709,E2 22094.709} C_VEL
LIN {X 0,Y 470.707,Z 622.298,A -85,B 0,C 180,E1 22092.767,E2 22092.767} C_VEL
LIN {X 0,Y 468.777,Z 638.966,A -85,B 0,C 180,E1 22090.407,E2 22090.407} C_VEL
LIN {X 0,Y 467.284,Z 652.645,A -85,B 0,C 180,E1 22088.113,E2 22088.113} C_VEL
LIN {X 0,Y 466.233,Z 663.623,A -85,B 0,C 180,E1 22085.988,E2 22085.988} C_VEL
LIN {X 0,Y 465.243,Z 675.459,A -85,B 0,C 180,E1 22083.279,E2 22083.279} C_VEL
LIN {X 0,Y 464.656,Z 683.882,A -85,B 0,C 180,E1 22080.95,E2 22080.95} C_VEL
LIN {X 0,Y 464.261,Z 691.491,A -85,B 0,C 180,E1 22078.422,E2 22078.422} C_VEL
LIN {X 0,Y 464.031,Z 697.651,A -85,B 0,C 180,E1 22075.752,E2 22075.752} C_VEL
LIN {X 0,Y 463.947,Z 701.812,A -85,B 0,C 180,E1 22073.352,E2 22073.352} C_VEL
LIN {X 0,Y 463.907,Z 704.913,A -85,B 0,C 180,E1 22070.7,E2 22070.7} C_VEL
LIN {X 0,Y 463.907,Z 706.277,A -85,B 0,C 180,E1 22068.081,E2 22068.081} C_VEL
LIN {X 0,Y 463.909,Z 706.262,A -85,B 0,C 180,E1 22065.758,E2 22065.758} C_VEL
LIN {X 0,Y 463.913,Z 704.794,A -85,B 0,C 180,E1 22063.08,E2 22063.08} C_VEL
LIN {X 0,Y 463.938,Z 701.807,A -85,B 0,C 180,E1 22060.556,E2 22060.556} C_VEL
LIN {X 0,Y 464.025,Z 697.689,A -85,B 0,C 180,E1 22058.176,E2 22058.176} C_VEL
LIN {X 0,Y 464.278,Z 691.343,A -85,B 0,C 180,E1 22055.438,E2 22055.438} C_VEL
LIN {X 0,Y 464.657,Z 683.883,A -85,B 0,C 180,E1 22052.96,E2 22052.96} C_VEL
LIN {X 0,Y 465.243,Z 675.403,A -85,B 0,C 180,E1 22050.616,E2 22050.616} C_VEL
LIN {X 0,Y 466.18,Z 664.166,A -85,B 0,C 180,E1 22048.034,E2 22048.034} C_VEL
LIN {X 0,Y 467.202,Z 653.484,A -85,B 0,C 180,E1 22045.95,E2 22045.95} C_VEL
LIN {X 0,Y 468.591,Z 640.553,A -85,B 0,C 180,E1 22043.753,E2 22043.753} C_VEL
LIN {X 0,Y 470.432,Z 624.518,A -85,B 0,C 180,E1 22041.444,E2 22041.444} C_VEL
LIN {X 0,Y 472.236,Z 610.202,A -85,B 0,C 180,E1 22039.632,E2 22039.632} C_VEL
LIN {X 0,Y 474.438,Z 592.346,A -85,B 0,C 180,E1 22037.711,E2 22037.711} C_VEL
LIN {X 0,Y 476.56,Z 574.652,A -85,B 0,C 180,E1 22036.1,E2 22036.1} C_VEL
LIN {X 0,Y 478.689,Z 555.149,A -85,B 0,C 180,E1 22034.617,E2 22034.617} C_VEL
LIN {X 0,Y 480.505,Z 536.298,A -85,B 0,C 180,E1 22033.437,E2 22033.437} C_VEL
LIN {X 0,Y 482.297,Z 514.86,A -85,B 0,C 180,E1 22032.351,E2 22032.351} C_VEL
LIN {X 0,Y 483.678,Z 494.134,A -85,B 0,C 180,E1 22031.535,E2 22031.535} C_VEL
LIN {X 0,Y 484.713,Z 472.435,A -85,B 0,C 180,E1 22030.916,E2 22030.916} C_VEL
LIN {X 0,Y 485.632,Z 437.586,A -85,B 0,C 180,E1 22030.278,E2 22030.278} C_VEL
LIN {X 0,Y 490.969,Z 224.631,A -85,B 0,C 180,E1 22026.614,E2 22026.614} C_VEL
LIN {X 0,Y 490.764,Z 223.181,A -85,B 0,C 180,E1 22026.564,E2 22026.564} C_VEL
LIN {X 0,Y 477.658,Z 203.199,A -85,B 0,C 180,E1 22024.763,E2 22024.763} C_VEL
LIN {X 0,Y 470.637,Z 193.243,A -85,B 0,C 180,E1 22023.769,E2 22023.769} C_VEL
LIN {X 0,Y 467.391,Z 188.579,A -85,B 0,C 180,E1 22023.284,E2 22023.284} C_VEL
LIN {X 0,Y 465.321,Z 185.222,A -85,B 0,C 180,E1 22022.554,E2 22022.554} C_VEL
LIN {X 0,Y 465.015,Z 183.814,A -85,B 0,C 180,E1 22022.326,E2 22022.326} C_VEL
LIN {X 0,Y 465.017,Z 183.802,A -85,B 0,C 180,E1 22018.608,E2 22018.608} C_VEL
LIN {X 0,Y 464.987,Z 183.803,A -85,B 0,C 180,E1 22014.962,E2 22014.962} C_VEL
LIN {X 0,Y 464.986,Z 183.804,A -85,B 0,C 180,E1 22011.313,E2 22011.313} C_VEL
LIN {X 0,Y 464.995,Z 183.802,A -85,B 0,C 180,E1 22007.699,E2 22007.699} C_VEL
LIN {X 0,Y 465.007,Z 183.799,A -85,B 0,C 180,E1 22003.989,E2 22003.989} C_VEL
LIN {X 0,Y 465.016,Z 183.796,A -85,B 0,C 180,E1 22000.331,E2 22000.331} C_VEL
LIN {X 0,Y 465.006,Z 183.798,A -85,B 0,C 180,E1 21996.676,E2 21996.676} C_VEL
LIN {X 0,Y 464.985,Z 183.805,A -85,B 0,C 180,E1 21992.959,E2 21992.959} C_VEL
LIN {X 0,Y 464.991,Z 183.817,A -85,B 0,C 180,E1 21989.358,E2 21989.358} C_VEL
LIN {X 0,Y 465.001,Z 183.81,A -85,B 0,C 180,E1 21985.717,E2 21985.717} C_VEL
LIN {X 0,Y 465.01,Z 183.797,A -85,B 0,C 180,E1 21982.069,E2 21982.069} C_VEL
LIN {X 0,Y 465.015,Z 183.797,A -85,B 0,C 180,E1 21978.426,E2 21978.426} C_VEL
LIN {X 0,Y 464.986,Z 183.813,A -85,B 0,C 180,E1 21974.827,E2 21974.827} C_VEL
LIN {X 0,Y 464.972,Z 183.816,A -85,B 0,C 180,E1 21971.159,E2 21971.159} C_VEL
LIN {X 0,Y 464.982,Z 183.807,A -85,B 0,C 180,E1 21967.538,E2 21967.538} C_VEL
LIN {X 0,Y 465,Z 183.797,A -85,B 0,C 180,E1 21963.879,E2 21963.879} C_VEL
LIN {X 0,Y 465.013,Z 183.799,A -85,B 0,C 180,E1 21960.247,E2 21960.247} C_VEL
LIN {X 0,Y 464.995,Z 183.808,A -85,B 0,C 180,E1 21956.672,E2 21956.672} C_VEL
LIN {X 0,Y 464.956,Z 183.818,A -85,B 0,C 180,E1 21953.084,E2 21953.084} C_VEL
LIN {X 0,Y 464.965,Z 183.817,A -85,B 0,C 180,E1 21949.468,E2 21949.468} C_VEL
LIN {X 0,Y 464.988,Z 183.813,A -85,B 0,C 180,E1 21945.811,E2 21945.811} C_VEL
LIN {X 0,Y 465.007,Z 183.804,A -85,B 0,C 180,E1 21942.093,E2 21942.093} C_VEL
LIN {X 0,Y 465.011,Z 183.8,A -85,B 0,C 180,E1 21938.428,E2 21938.428} C_VEL
LIN {X 0,Y 465.028,Z 183.941,A -85,B 0,C 180,E1 21935.99,E2 21935.99} C_VEL
LIN {X 0,Y 466.283,Z 187.301,A -85,B 0,C 180,E1 21935.418,E2 21935.418} C_VEL
LIN {X 0,Y 467.409,Z 188.841,A -85,B 0,C 180,E1 21935.077,E2 21935.077} C_VEL
LIN {X 0,Y 469.318,Z 192.668,A -85,B 0,C 180,E1 21934.375,E2 21934.375} C_VEL
LIN {X 0,Y 477.234,Z 208.453,A -85,B 0,C 180,E1 21931.603,E2 21931.603} C_VEL
LIN {X 0,Y 485.428,Z 225.496,A -85,B 0,C 180,E1 21928.869,E2 21928.869} C_VEL
LIN {X 0,Y 491.238,Z 238.643,A -85,B 0,C 180,E1 21926.943,E2 21926.943} C_VEL
LIN {X 0,Y 488.113,Z 279.082,A -85,B 0,C 180,E1 21923.613,E2 21923.613} C_VEL
LIN {X 0,Y 487.005,Z 302.997,A -85,B 0,C 180,E1 21921.615,E2 21921.615} C_VEL
LIN {X 0,Y 488.113,Z 319.973,A -85,B 0,C 180,E1 21920.038,E2 21920.038} C_VEL
LIN {X 0,Y 491.017,Z 334.551,A -85,B 0,C 180,E1 21918.535,E2 21918.535} C_VEL
LIN {X 0,Y 495.394,Z 347.103,A -85,B 0,C 180,E1 21917.109,E2 21917.109} C_VEL
LIN {X 0,Y 501.757,Z 358.887,A -85,B 0,C 180,E1 21915.618,E2 21915.618} C_VEL
LIN {X 0,Y 509.968,Z 369.205,A -85,B 0,C 180,E1 21914.145,E2 21914.145} C_VEL
LIN {X 0,Y 519.27,Z 377.439,A -85,B 0,C 180,E1 21912.81,E2 21912.81} C_VEL
LIN {X 0,Y 529.509,Z 383.948,A -85,B 0,C 180,E1 21911.604,E2 21911.604} C_VEL
LIN {X 0,Y 541.729,Z 389.357,A -85,B 0,C 180,E1 21910.41,E2 21910.41} C_VEL
LIN {X 0,Y 541.693,Z 389.785,A -85,B 0,C 180,E1 21910.382,E2 21910.382} C_VEL
LIN {X 0,Y 521.611,Z 416.742,A -85,B 0,C 180,E1 21909.731,E2 21909.731} C_VEL
LIN {X 0,Y 512.082,Z 431.718,A -85,B 0,C 180,E1 21909.244,E2 21909.244} C_VEL
LIN {X 0,Y 505.14,Z 444.803,A -85,B 0,C 180,E1 21908.717,E2 21908.717} C_VEL
LIN {X 0,Y 497.213,Z 458.494,A -85,B 0,C 180,E1 21908.196,E2 21908.196} C_VEL
LIN {X 0,Y 491.669,Z 471.08,A -85,B 0,C 180,E1 21907.595,E2 21907.595} C_VEL
LIN {X 0,Y 487.448,Z 481.313,A -85,B 0,C 180,E1 21907.114,E2 21907.114} C_VEL
LIN {X 0,Y 486.318,Z 496.648,A -85,B 0,C 180,E1 21906.936,E2 21906.936} C_VEL
LIN {X 0,Y 485.414,Z 527.384,A -85,B 0,C 180,E1 21906.381,E2 21906.381} C_VEL
LIN {X 0,Y 483.989,Z 551.071,A -85,B 0,C 180,E1 21905.751,E2 21905.751} C_VEL
LIN {X 0,Y 482.343,Z 573.318,A -85,B 0,C 180,E1 21904.935,E2 21904.935} C_VEL
LIN {X 0,Y 480.603,Z 594.109,A -85,B 0,C 180,E1 21903.964,E2 21903.964} C_VEL
LIN {X 0,Y 478.68,Z 615.17,A -85,B 0,C 180,E1 21902.751,E2 21902.751} C_VEL
LIN {X 0,Y 476.743,Z 634.805,A -85,B 0,C 180,E1 21901.396,E2 21901.396} C_VEL
LIN {X 0,Y 474.82,Z 653.627,A -85,B 0,C 180,E1 21899.862,E2 21899.862} C_VEL
LIN {X 0,Y 472.887,Z 671.759,A -85,B 0,C 180,E1 21898.132,E2 21898.132} C_VEL
LIN {X 0,Y 471.041,Z 689.079,A -85,B 0,C 180,E1 21896.2,E2 21896.2} C_VEL
LIN {X 0,Y 469.399,Z 703.534,A -85,B 0,C 180,E1 21894.263,E2 21894.263} C_VEL
LIN {X 0,Y 467.748,Z 718.394,A -85,B 0,C 180,E1 21891.919,E2 21891.919} C_VEL
LIN {X 0,Y 466.456,Z 731.227,A -85,B 0,C 180,E1 21889.535,E2 21889.535} C_VEL
LIN {X 0,Y 465.47,Z 742.416,A -85,B 0,C 180,E1 21887.083,E2 21887.083} C_VEL
LIN {X 0,Y 464.75,Z 752.421,A -85,B 0,C 180,E1 21884.451,E2 21884.451} C_VEL
LIN {X 0,Y 464.287,Z 760.929,A -85,B 0,C 180,E1 21881.679,E2 21881.679} C_VEL
LIN {X 0,Y 464.039,Z 767.457,A -85,B 0,C 180,E1 21878.925,E2 21878.925} C_VEL
LIN {X 0,Y 463.941,Z 772.168,A -85,B 0,C 180,E1 21876.186,E2 21876.186} C_VEL
LIN {X 0,Y 463.911,Z 775.034,A -85,B 0,C 180,E1 21873.583,E2 21873.583} C_VEL
LIN {X 0,Y 463.907,Z 776.399,A -85,B 0,C 180,E1 21870.864,E2 21870.864} C_VEL
LIN {X 0,Y 463.904,Z 776.109,A -85,B 0,C 180,E1 21868.147,E2 21868.147} C_VEL
LIN {X 0,Y 463.919,Z 774.246,A -85,B 0,C 180,E1 21865.55,E2 21865.55} C_VEL
LIN {X 0,Y 463.972,Z 770.854,A -85,B 0,C 180,E1 21862.944,E2 21862.944} C_VEL
LIN {X 0,Y 464.094,Z 765.593,A -85,B 0,C 180,E1 21860.2,E2 21860.2} C_VEL
LIN {X 0,Y 464.407,Z 758.43,A -85,B 0,C 180,E1 21857.44,E2 21857.44} C_VEL
LIN {X 0,Y 464.932,Z 749.723,A -85,B 0,C 180,E1 21854.789,E2 21854.789} C_VEL
LIN {X 0,Y 465.713,Z 739.558,A -85,B 0,C 180,E1 21852.25,E2 21852.25} C_VEL
LIN {X 0,Y 466.817,Z 727.549,A -85,B 0,C 180,E1 21849.74,E2 21849.74} C_VEL
LIN {X 0,Y 468.194,Z 714.291,A -85,B 0,C 180,E1 21847.393,E2 21847.393} C_VEL
LIN {X 0,Y 469.928,Z 698.95,A -85,B 0,C 180,E1 21845.084,E2 21845.084} C_VEL
LIN {X 0,Y 471.422,Z 685.41,A -85,B 0,C 180,E1 21843.37,E2 21843.37} C_VEL
LIN {X 0,Y 473.279,Z 667.723,A -85,B 0,C 180,E1 21841.481,E2 21841.481} C_VEL
LIN {X 0,Y 475.295,Z 647.773,A -85,B 0,C 180,E1 21839.676,E2 21839.676} C_VEL
LIN {X 0,Y 477.282,Z 627.577,A -85,B 0,C 180,E1 21838.135,E2 21838.135} C_VEL
LIN {X 0,Y 479.186,Z 606.459,A -85,B 0,C 180,E1 21836.795,E2 21836.795} C_VEL
LIN {X 0,Y 481.053,Z 584.364,A -85,B 0,C 180,E1 21835.645,E2 21835.645} C_VEL
LIN {X 0,Y 482.756,Z 561.884,A -85,B 0,C 180,E1 21834.705,E2 21834.705} C_VEL
LIN {X 0,Y 484.26,Z 539.175,A -85,B 0,C 180,E1 21833.994,E2 21833.994} C_VEL
LIN {X 0,Y 485.465,Z 514.163,A -85,B 0,C 180,E1 21833.438,E2 21833.438} C_VEL
LIN {X 0,Y 486.315,Z 484.966,A -85,B 0,C 180,E1 21832.978,E2 21832.978} C_VEL
LIN {X 0,Y 486.965,Z 475.866,A -85,B 0,C 180,E1 21832.868,E2 21832.868} C_VEL
LIN {X 0,Y 494.879,Z 446.699,A -85,B 0,C 180,E1 21831.811,E2 21831.811} C_VEL
LIN {X 0,Y 500.676,Z 430.2,A -85,B 0,C 180,E1 21831.313,E2 21831.313} C_VEL
LIN {X 0,Y 505.788,Z 413.359,A -85,B 0,C 180,E1 21830.758,E2 21830.758} C_VEL
LIN {X 0,Y 514.05,Z 392.441,A -85,B 0,C 180,E1 21830.213,E2 21830.213} C_VEL
LIN {X 0,Y 527.319,Z 364.047,A -85,B 0,C 180,E1 21829.637,E2 21829.637} C_VEL
LIN {X 0,Y 533.958,Z 350.739,A -85,B 0,C 180,E1 21829.405,E2 21829.405} C_VEL
LIN {X 0,Y 539.197,Z 335.255,A -85,B 0,C 180,E1 21828.971,E2 21828.971} C_VEL
LIN {X 0,Y 550.465,Z 308.771,A -85,B 0,C 180,E1 21828.402,E2 21828.402} C_VEL
LIN {X 0,Y 554.297,Z 299.99,A -85,B 0,C 180,E1 21828.225,E2 21828.225} C_VEL
LIN {X 0,Y 542.709,Z 295.17,A -85,B 0,C 180,E1 21827.16,E2 21827.16} C_VEL
LIN {X 0,Y 532.11,Z 288.825,A -85,B 0,C 180,E1 21826.027,E2 21826.027} C_VEL
LIN {X 0,Y 518.307,Z 277.999,A -85,B 0,C 180,E1 21824.293,E2 21824.293} C_VEL
LIN {X 0,Y 509.523,Z 268.212,A -85,B 0,C 180,E1 21822.916,E2 21822.916} C_VEL
LIN {X 0,Y 503.377,Z 258.53,A -85,B 0,C 180,E1 21821.713,E2 21821.713} C_VEL
LIN {X 0,Y 491.04,Z 231.334,A -85,B 0,C 180,E1 21818.541,E2 21818.541} C_VEL
LIN {X 0,Y 483.243,Z 215.923,A -85,B 0,C 180,E1 21816.428,E2 21816.428} C_VEL
LIN {X 0,Y 476.663,Z 204.06,A -85,B 0,C 180,E1 21814.569,E2 21814.569} C_VEL
LIN {X 0,Y 474.205,Z 204.876,A -85,B 0,C 180,E1 21814.261,E2 21814.261} C_VEL
LIN {X 0,Y 472.587,Z 204.579,A -85,B 0,C 180,E1 21813.955,E2 21813.955} C_VEL
LIN {X 0,Y 473.29,Z 241.127,A -85,B 0,C 180,E1 21811.17,E2 21811.17} C_VEL
LIN {X 0,Y 473.588,Z 275.992,A -85,B 0,C 180,E1 21808.361,E2 21808.361} C_VEL
LIN {X 0,Y 473.421,Z 309.916,A -85,B 0,C 180,E1 21805.521,E2 21805.521} C_VEL
LIN {X 0,Y 473.009,Z 332.125,A -85,B 0,C 180,E1 21803.613,E2 21803.613} C_VEL
LIN {X 0,Y 472.133,Z 336.54,A -85,B 0,C 180,E1 21803.335,E2 21803.335} C_VEL
LIN {X 0,Y 470.155,Z 447.4,A -85,B 0,C 180,E1 21801.344,E2 21801.344} C_VEL
LIN {X 0,Y 469.795,Z 501.777,A -85,B 0,C 180,E1 21800.412,E2 21800.412} C_VEL
LIN {X 0,Y 469.725,Z 519.044,A -85,B 0,C 180,E1 21799.903,E2 21799.903} C_VEL
LIN {X 0,Y 469.472,Z 535.062,A -85,B 0,C 180,E1 21799.211,E2 21799.211} C_VEL
LIN {X 0,Y 469.058,Z 551.452,A -85,B 0,C 180,E1 21798.261,E2 21798.261} C_VEL
LIN {X 0,Y 468.564,Z 565.835,A -85,B 0,C 180,E1 21797.19,E2 21797.19} C_VEL
LIN {X 0,Y 467.952,Z 579.863,A -85,B 0,C 180,E1 21795.872,E2 21795.872} C_VEL
LIN {X 0,Y 467.32,Z 592.74,A -85,B 0,C 180,E1 21794.37,E2 21794.37} C_VEL
LIN {X 0,Y 466.71,Z 603.93,A -85,B 0,C 180,E1 21792.748,E2 21792.748} C_VEL
LIN {X 0,Y 466.164,Z 613.531,A -85,B 0,C 180,E1 21791.004,E2 21791.004} C_VEL
LIN {X 0,Y 465.726,Z 621.679,A -85,B 0,C 180,E1 21789.141,E2 21789.141} C_VEL
LIN {X 0,Y 465.376,Z 628.317,A -85,B 0,C 180,E1 21787.158,E2 21787.158} C_VEL
LIN {X 0,Y 465.122,Z 633.032,A -85,B 0,C 180,E1 21785.18,E2 21785.18} C_VEL
LIN {X 0,Y 464.949,Z 636.373,A -85,B 0,C 180,E1 21782.958,E2 21782.958} C_VEL
LIN {X 0,Y 464.862,Z 637.753,A -85,B 0,C 180,E1 21780.862,E2 21780.862} C_VEL
LIN {X 0,Y 464.826,Z 637.373,A -85,B 0,C 180,E1 21778.767,E2 21778.767} C_VEL
LIN {X 0,Y 464.848,Z 635.142,A -85,B 0,C 180,E1 21776.547,E2 21776.547} C_VEL
LIN {X 0,Y 464.948,Z 631.264,A -85,B 0,C 180,E1 21774.446,E2 21774.446} C_VEL
LIN {X 0,Y 465.147,Z 625.429,A -85,B 0,C 180,E1 21772.341,E2 21772.341} C_VEL
LIN {X 0,Y 465.462,Z 618.037,A -85,B 0,C 180,E1 21770.354,E2 21770.354} C_VEL
LIN {X 0,Y 465.89,Z 609.157,A -85,B 0,C 180,E1 21768.487,E2 21768.487} C_VEL
LIN {X 0,Y 466.438,Z 598.478,A -85,B 0,C 180,E1 21766.706,E2 21766.706} C_VEL
LIN {X 0,Y 467.092,Z 586.233,A -85,B 0,C 180,E1 21765.052,E2 21765.052} C_VEL
LIN {X 0,Y 467.768,Z 573.139,A -85,B 0,C 180,E1 21763.611,E2 21763.611} C_VEL
LIN {X 0,Y 468.449,Z 558.225,A -85,B 0,C 180,E1 21762.292,E2 21762.292} C_VEL
LIN {X 0,Y 469.068,Z 543.114,A -85,B 0,C 180,E1 21761.223,E2 21761.223} C_VEL
LIN {X 0,Y 469.595,Z 526.541,A -85,B 0,C 180,E1 21760.309,E2 21760.309} C_VEL
LIN {X 0,Y 469.996,Z 509.059,A -85,B 0,C 180,E1 21759.609,E2 21759.609} C_VEL
LIN {X 0,Y 470.207,Z 490.987,A -85,B 0,C 180,E1 21759.126,E2 21759.126} C_VEL
LIN {X 0,Y 472.247,Z 329.881,A -85,B 0,C 180,E1 21756.403,E2 21756.403} C_VEL
LIN {X 0,Y 471.395,Z 324.337,A -85,B 0,C 180,E1 21756.234,E2 21756.234} C_VEL
LIN {X 0,Y 472.423,Z 287.324,A -85,B 0,C 180,E1 21752.737,E2 21752.737} C_VEL
LIN {X 0,Y 473.369,Z 250.46,A -85,B 0,C 180,E1 21749.259,E2 21749.259} C_VEL
LIN {X 0,Y 473.576,Z 243.879,A -85,B 0,C 180,E1 21748.603,E2 21748.603} C_VEL
LIN {X 0,Y 475.12,Z 245.347,A -85,B 0,C 180,E1 21748.398,E2 21748.398} C_VEL
LIN {X 0,Y 477.434,Z 245.324,A -85,B 0,C 180,E1 21748.146,E2 21748.146} C_VEL
LIN {X 0,Y 480.777,Z 243.203,A -85,B 0,C 180,E1 21747.832,E2 21747.832} C_VEL
LIN {X 0,Y 482.064,Z 242.133,A -85,B 0,C 180,E1 21747.718,E2 21747.718} C_VEL
LIN {X 0,Y 486.035,Z 241.71,A -85,B 0,C 180,E1 21747.315,E2 21747.315} C_VEL
LIN {X 0,Y 490.014,Z 239.837,A -85,B 0,C 180,E1 21746.955,E2 21746.955} C_VEL
LIN {X 0,Y 488.142,Z 316.969,A -85,B 0,C 180,E1 21745.631,E2 21745.631} C_VEL
LIN {X 0,Y 487.136,Z 324.66,A -85,B 0,C 180,E1 21745.574,E2 21745.574} C_VEL
LIN {X 0,Y 481.681,Z 345.179,A -85,B 0,C 180,E1 21745.674,E2 21745.674} C_VEL
LIN {X 0,Y 480.936,Z 351.773,A -85,B 0,C 180,E1 21745.612,E2 21745.612} C_VEL
LIN {X 0,Y 477.821,Z 473.095,A -85,B 0,C 180,E1 21743.473,E2 21743.473} C_VEL
LIN {X 0,Y 476.802,Z 494.628,A -85,B 0,C 180,E1 21742.865,E2 21742.865} C_VEL
LIN {X 0,Y 475.46,Z 515.416,A -85,B 0,C 180,E1 21742.055,E2 21742.055} C_VEL
LIN {X 0,Y 473.844,Z 535.105,A -85,B 0,C 180,E1 21741.076,E2 21741.076} C_VEL
LIN {X 0,Y 471.941,Z 554.229,A -85,B 0,C 180,E1 21739.891,E2 21739.891} C_VEL
LIN {X 0,Y 469.873,Z 572.645,A -85,B 0,C 180,E1 21738.507,E2 21738.507} C_VEL
LIN {X 0,Y 467.649,Z 590.648,A -85,B 0,C 180,E1 21736.899,E2 21736.899} C_VEL
LIN {X 0,Y 465.411,Z 607.999,A -85,B 0,C 180,E1 21735.063,E2 21735.063} C_VEL
LIN {X 0,Y 463.275,Z 623.746,A -85,B 0,C 180,E1 21733.085,E2 21733.085} C_VEL
LIN {X 0,Y 461.324,Z 638.77,A -85,B 0,C 180,E1 21730.886,E2 21730.886} C_VEL
LIN {X 0,Y 459.415,Z 654.298,A -85,B 0,C 180,E1 21728.177,E2 21728.177} C_VEL
LIN {X 0,Y 458.196,Z 666.436,A -85,B 0,C 180,E1 21725.73,E2 21725.73} C_VEL
LIN {X 0,Y 457.282,Z 676.514,A -85,B 0,C 180,E1 21723.286,E2 21723.286} C_VEL
LIN {X 0,Y 456.686,Z 684.645,A -85,B 0,C 180,E1 21720.965,E2 21720.965} C_VEL
LIN {X 0,Y 456.231,Z 692.75,A -85,B 0,C 180,E1 21718.112,E2 21718.112} C_VEL
LIN {X 0,Y 456.033,Z 698.061,A -85,B 0,C 180,E1 21715.693,E2 21715.693} C_VEL
LIN {X 0,Y 455.947,Z 702.141,A -85,B 0,C 180,E1 21713.242,E2 21713.242} C_VEL
LIN {X 0,Y 455.912,Z 705.152,A -85,B 0,C 180,E1 21710.408,E2 21710.408} C_VEL
LIN {X 0,Y 455.907,Z 706.294,A -85,B 0,C 180,E1 21708.013,E2 21708.013} C_VEL
LIN {X 0,Y 455.905,Z 706.242,A -85,B 0,C 180,E1 21705.65,E2 21705.65} C_VEL
LIN {X 0,Y 455.914,Z 704.72,A -85,B 0,C 180,E1 21702.926,E2 21702.926} C_VEL
LIN {X 0,Y 455.946,Z 701.679,A -85,B 0,C 180,E1 21700.36,E2 21700.36} C_VEL
LIN {X 0,Y 456.05,Z 697.529,A -85,B 0,C 180,E1 21697.939,E2 21697.939} C_VEL
LIN {X 0,Y 456.317,Z 691.124,A -85,B 0,C 180,E1 21695.154,E2 21695.154} C_VEL
LIN {X 0,Y 456.743,Z 683.626,A -85,B 0,C 180,E1 21692.635,E2 21692.635} C_VEL
LIN {X 0,Y 457.392,Z 675.114,A -85,B 0,C 180,E1 21690.251,E2 21690.251} C_VEL
LIN {X 0,Y 458.426,Z 663.804,A -85,B 0,C 180,E1 21687.625,E2 21687.625} C_VEL
LIN {X 0,Y 459.557,Z 653.083,A -85,B 0,C 180,E1 21685.508,E2 21685.508} C_VEL
LIN {X 0,Y 461.415,Z 637.973,A -85,B 0,C 180,E1 21682.905,E2 21682.905} C_VEL
LIN {X 0,Y 463.284,Z 623.623,A -85,B 0,C 180,E1 21680.81,E2 21680.81} C_VEL
LIN {X 0,Y 465.482,Z 607.366,A -85,B 0,C 180,E1 21678.778,E2 21678.778} C_VEL
LIN {X 0,Y 467.629,Z 590.819,A -85,B 0,C 180,E1 21677.026,E2 21677.026} C_VEL
LIN {X 0,Y 469.905,Z 572.656,A -85,B 0,C 180,E1 21675.396,E2 21675.396} C_VEL
LIN {X 0,Y 472.058,Z 553.709,A -85,B 0,C 180,E1 21673.969,E2 21673.969} C_VEL
LIN {X 0,Y 474.039,Z 534.218,A -85,B 0,C 180,E1 21672.762,E2 21672.762} C_VEL
LIN {X 0,Y 475.7,Z 514.491,A -85,B 0,C 180,E1 21671.781,E2 21671.781} C_VEL
LIN {X 0,Y 477.111,Z 493.424,A -85,B 0,C 180,E1 21670.962,E2 21670.962} C_VEL
LIN {X 0,Y 478.18,Z 472,A -85,B 0,C 180,E1 21670.355,E2 21670.355} C_VEL
LIN {X 0,Y 480.608,Z 380.568,A -85,B 0,C 180,E1 21668.73,E2 21668.73} C_VEL
LIN {X 0,Y 484.798,Z 226.754,A -85,B 0,C 180,E1 21666.016,E2 21666.016} C_VEL
LIN {X 0,Y 472.202,Z 207.749,A -85,B 0,C 180,E1 21664.252,E2 21664.252} C_VEL
LIN {X 0,Y 464.642,Z 197.008,A -85,B 0,C 180,E1 21663.156,E2 21663.156} C_VEL
LIN {X 0,Y 462.089,Z 193.954,A -85,B 0,C 180,E1 21662.788,E2 21662.788} C_VEL
LIN {X 0,Y 460.355,Z 191.925,A -85,B 0,C 180,E1 21662.529,E2 21662.529} C_VEL
LIN {X 0,Y 459.412,Z 189.519,A -85,B 0,C 180,E1 21662.082,E2 21662.082} C_VEL
LIN {X 0,Y 457.492,Z 186.59,A -85,B 0,C 180,E1 21661.404,E2 21661.404} C_VEL
LIN {X 0,Y 457.063,Z 184.79,A -85,B 0,C 180,E1 21661.089,E2 21661.089} C_VEL
LIN {X 0,Y 457.031,Z 184.798,A -85,B 0,C 180,E1 21657.44,E2 21657.44} C_VEL
LIN {X 0,Y 457.011,Z 184.807,A -85,B 0,C 180,E1 21653.793,E2 21653.793} C_VEL
LIN {X 0,Y 457.036,Z 184.805,A -85,B 0,C 180,E1 21650.134,E2 21650.134} C_VEL
LIN {X 0,Y 457.063,Z 184.801,A -85,B 0,C 180,E1 21646.442,E2 21646.442} C_VEL
LIN {X 0,Y 457.073,Z 184.799,A -85,B 0,C 180,E1 21642.692,E2 21642.692} C_VEL
LIN {X 0,Y 457.054,Z 184.799,A -85,B 0,C 180,E1 21639.05,E2 21639.05} C_VEL
LIN {X 0,Y 457.02,Z 184.8,A -85,B 0,C 180,E1 21635.434,E2 21635.434} C_VEL
LIN {X 0,Y 457.018,Z 184.79,A -85,B 0,C 180,E1 21631.673,E2 21631.673} C_VEL
LIN {X 0,Y 457.044,Z 184.792,A -85,B 0,C 180,E1 21628.057,E2 21628.057} C_VEL
LIN {X 0,Y 457.069,Z 184.799,A -85,B 0,C 180,E1 21624.422,E2 21624.422} C_VEL
LIN {X 0,Y 457.07,Z 184.799,A -85,B 0,C 180,E1 21620.756,E2 21620.756} C_VEL
LIN {X 0,Y 457.042,Z 184.796,A -85,B 0,C 180,E1 21617.057,E2 21617.057} C_VEL
LIN {X 0,Y 457.009,Z 184.79,A -85,B 0,C 180,E1 21613.539,E2 21613.539} C_VEL
LIN {X 0,Y 457.028,Z 184.8,A -85,B 0,C 180,E1 21609.826,E2 21609.826} C_VEL
LIN {X 0,Y 457.056,Z 184.801,A -85,B 0,C 180,E1 21606.154,E2 21606.154} C_VEL
LIN {X 0,Y 457.073,Z 184.799,A -85,B 0,C 180,E1 21602.508,E2 21602.508} C_VEL
LIN {X 0,Y 457.054,Z 184.797,A -85,B 0,C 180,E1 21598.872,E2 21598.872} C_VEL
LIN {X 0,Y 457.024,Z 184.794,A -85,B 0,C 180,E1 21595.232,E2 21595.232} C_VEL
LIN {X 0,Y 457.009,Z 184.795,A -85,B 0,C 180,E1 21591.445,E2 21591.445} C_VEL
LIN {X 0,Y 457.038,Z 184.793,A -85,B 0,C 180,E1 21587.749,E2 21587.749} C_VEL
LIN {X 0,Y 457.064,Z 184.793,A -85,B 0,C 180,E1 21584.131,E2 21584.131} C_VEL
LIN {X 0,Y 457.073,Z 184.801,A -85,B 0,C 180,E1 21580.447,E2 21580.447} C_VEL
LIN {X 0,Y 457.058,Z 184.915,A -85,B 0,C 180,E1 21577.159,E2 21577.159} C_VEL
LIN {X 0,Y 458.23,Z 188.075,A -85,B 0,C 180,E1 21576.602,E2 21576.602} C_VEL
LIN {X 0,Y 459.646,Z 190.189,A -85,B 0,C 180,E1 21576.134,E2 21576.134} C_VEL
LIN {X 0,Y 461.722,Z 194.11,A -85,B 0,C 180,E1 21575.364,E2 21575.364} C_VEL
LIN {X 0,Y 468.986,Z 208.632,A -85,B 0,C 180,E1 21572.718,E2 21572.718} C_VEL
LIN {X 0,Y 477.072,Z 225.234,A -85,B 0,C 180,E1 21569.941,E2 21569.941} C_VEL
LIN {X 0,Y 484.833,Z 242.294,A -85,B 0,C 180,E1 21567.343,E2 21567.343} C_VEL
LIN {X 0,Y 481.427,Z 283.815,A -85,B 0,C 180,E1 21563.891,E2 21563.891} C_VEL
LIN {X 0,Y 480.382,Z 306.469,A -85,B 0,C 180,E1 21561.969,E2 21561.969} C_VEL
LIN {X 0,Y 481.455,Z 323.26,A -85,B 0,C 180,E1 21560.39,E2 21560.39} C_VEL
LIN {X 0,Y 484.391,Z 338.336,A -85,B 0,C 180,E1 21558.817,E2 21558.817} C_VEL
LIN {X 0,Y 489.092,Z 351.88,A -85,B 0,C 180,E1 21557.257,E2 21557.257} C_VEL
LIN {X 0,Y 495.555,Z 363.856,A -85,B 0,C 180,E1 21555.725,E2 21555.725} C_VEL
LIN {X 0,Y 503.746,Z 374.261,A -85,B 0,C 180,E1 21554.232,E2 21554.232} C_VEL
LIN {X 0,Y 512.988,Z 382.651,A -85,B 0,C 180,E1 21552.874,E2 21552.874} C_VEL
LIN {X 0,Y 523.134,Z 389.366,A -85,B 0,C 180,E1 21551.642,E2 21551.642} C_VEL
LIN {X 0,Y 531.27,Z 393.501,A -85,B 0,C 180,E1 21550.79,E2 21550.79} C_VEL
LIN {X 0,Y 514.751,Z 415.94,A -85,B 0,C 180,E1 21550.238,E2 21550.238} C_VEL
LIN {X 0,Y 505.217,Z 431.154,A -85,B 0,C 180,E1 21549.735,E2 21549.735} C_VEL
LIN {X 0,Y 498.646,Z 443.416,A -85,B 0,C 180,E1 21549.244,E2 21549.244} C_VEL
LIN {X 0,Y 490.74,Z 457.129,A -85,B 0,C 180,E1 21548.719,E2 21548.719} C_VEL
LIN {X 0,Y 485.122,Z 469.705,A -85,B 0,C 180,E1 21548.118,E2 21548.118} C_VEL
LIN {X 0,Y 481.41,Z 478.621,A -85,B 0,C 180,E1 21547.709,E2 21547.709} C_VEL
LIN {X 0,Y 479.945,Z 495.983,A -85,B 0,C 180,E1 21547.522,E2 21547.522} C_VEL
LIN {X 0,Y 479.01,Z 525.367,A -85,B 0,C 180,E1 21546.981,E2 21546.981} C_VEL
LIN {X 0,Y 477.426,Z 549.318,A -85,B 0,C 180,E1 21546.34,E2 21546.34} C_VEL
LIN {X 0,Y 475.639,Z 571.875,A -85,B 0,C 180,E1 21545.504,E2 21545.504} C_VEL
LIN {X 0,Y 473.629,Z 593.974,A -85,B 0,C 180,E1 21544.455,E2 21544.455} C_VEL
LIN {X 0,Y 471.487,Z 615.788,A -85,B 0,C 180,E1 21543.17,E2 21543.17} C_VEL
LIN {X 0,Y 469.359,Z 635.839,A -85,B 0,C 180,E1 21541.747,E2 21541.747} C_VEL
LIN {X 0,Y 467.316,Z 654.448,A -85,B 0,C 180,E1 21540.185,E2 21540.185} C_VEL
LIN {X 0,Y 465.213,Z 673.134,A -85,B 0,C 180,E1 21538.358,E2 21538.358} C_VEL
LIN {X 0,Y 463.09,Z 691.685,A -85,B 0,C 180,E1 21536.202,E2 21536.202} C_VEL
LIN {X 0,Y 461.32,Z 707.457,A -85,B 0,C 180,E1 21534.046,E2 21534.046} C_VEL
LIN {X 0,Y 459.966,Z 719.629,A -85,B 0,C 180,E1 21532.09,E2 21532.09} C_VEL
LIN {X 0,Y 458.513,Z 733.13,A -85,B 0,C 180,E1 21529.49,E2 21529.49} C_VEL
LIN {X 0,Y 457.415,Z 744.904,A -85,B 0,C 180,E1 21526.77,E2 21526.77} C_VEL
LIN {X 0,Y 456.674,Z 754.947,A -85,B 0,C 180,E1 21523.936,E2 21523.936} C_VEL
LIN {X 0,Y 456.228,Z 762.897,A -85,B 0,C 180,E1 21521.119,E2 21521.119} C_VEL
LIN {X 0,Y 456.019,Z 768.914,A -85,B 0,C 180,E1 21518.32,E2 21518.32} C_VEL
LIN {X 0,Y 455.936,Z 772.98,A -85,B 0,C 180,E1 21515.663,E2 21515.663} C_VEL
LIN {X 0,Y 455.913,Z 775.576,A -85,B 0,C 180,E1 21512.891,E2 21512.891} C_VEL
LIN {X 0,Y 455.909,Z 776.489,A -85,B 0,C 180,E1 21510.125,E2 21510.125} C_VEL
LIN {X 0,Y 455.909,Z 775.783,A -85,B 0,C 180,E1 21507.486,E2 21507.486} C_VEL
LIN {X 0,Y 455.93,Z 773.591,A -85,B 0,C 180,E1 21504.841,E2 21504.841} C_VEL
LIN {X 0,Y 456.003,Z 769.602,A -85,B 0,C 180,E1 21502.06,E2 21502.06} C_VEL
LIN {X 0,Y 456.191,Z 763.813,A -85,B 0,C 180,E1 21499.263,E2 21499.263} C_VEL
LIN {X 0,Y 456.57,Z 756.524,A -85,B 0,C 180,E1 21496.577,E2 21496.577} C_VEL
LIN {X 0,Y 457.177,Z 747.853,A -85,B 0,C 180,E1 21494.004,E2 21494.004} C_VEL
LIN {X 0,Y 458.164,Z 736.696,A -85,B 0,C 180,E1 21491.284,E2 21491.284} C_VEL
LIN {X 0,Y 459.483,Z 723.922,A -85,B 0,C 180,E1 21488.691,E2 21488.691} C_VEL
LIN {X 0,Y 460.848,Z 711.724,A -85,B 0,C 180,E1 21486.597,E2 21486.597} C_VEL
LIN {X 0,Y 462.503,Z 696.607,A -85,B 0,C 180,E1 21484.455,E2 21484.455} C_VEL
LIN {X 0,Y 464.361,Z 679.85,A -85,B 0,C 180,E1 21482.423,E2 21482.423} C_VEL
LIN {X 0,Y 466.303,Z 662.208,A -85,B 0,C 180,E1 21480.592,E2 21480.592} C_VEL
LIN {X 0,Y 468.416,Z 642.551,A -85,B 0,C 180,E1 21478.865,E2 21478.865} C_VEL
LIN {X 0,Y 470.494,Z 621.837,A -85,B 0,C 180,E1 21477.331,E2 21477.331} C_VEL
LIN {X 0,Y 472.547,Z 601.079,A -85,B 0,C 180,E1 21476.04,E2 21476.04} C_VEL
LIN {X 0,Y 474.475,Z 578.865,A -85,B 0,C 180,E1 21474.916,E2 21474.916} C_VEL
LIN {X 0,Y 476.416,Z 554.877,A -85,B 0,C 180,E1 21473.964,E2 21473.964} C_VEL
LIN {X 0,Y 478.011,Z 532.033,A -85,B 0,C 180,E1 21473.28,E2 21473.28} C_VEL
LIN {X 0,Y 479.095,Z 507.751,A -85,B 0,C 180,E1 21472.774,E2 21472.774} C_VEL
LIN {X 0,Y 479.879,Z 484.508,A -85,B 0,C 180,E1 21472.415,E2 21472.415} C_VEL
LIN {X 0,Y 480.987,Z 471.728,A -85,B 0,C 180,E1 21472.251,E2 21472.251} C_VEL
LIN {X 0,Y 488.423,Z 445.057,A -85,B 0,C 180,E1 21471.288,E2 21471.288} C_VEL
LIN {X 0,Y 493.882,Z 429.766,A -85,B 0,C 180,E1 21470.828,E2 21470.828} C_VEL
LIN {X 0,Y 499.008,Z 412.923,A -85,B 0,C 180,E1 21470.269,E2 21470.269} C_VEL
LIN {X 0,Y 507.241,Z 392.009,A -85,B 0,C 180,E1 21469.718,E2 21469.718} C_VEL
LIN {X 0,Y 519.865,Z 364.85,A -85,B 0,C 180,E1 21469.162,E2 21469.162} C_VEL
LIN {X 0,Y 527.654,Z 349.174,A -85,B 0,C 180,E1 21468.887,E2 21468.887} C_VEL
LIN {X 0,Y 533.435,Z 332.545,A -85,B 0,C 180,E1 21468.43,E2 21468.43} C_VEL
LIN {X 0,Y 545.127,Z 304.997,A -85,B 0,C 180,E1 21467.839,E2 21467.839} C_VEL
LIN {X 0,Y 532.611,Z 298.723,A -85,B 0,C 180,E1 21466.594,E2 21466.594} C_VEL
LIN {X 0,Y 517.122,Z 287.51,A -85,B 0,C 180,E1 21464.732,E2 21464.732} C_VEL
LIN {X 0,Y 508.534,Z 279.282,A -85,B 0,C 180,E1 21463.484,E2 21463.484} C_VEL
LIN {X 0,Y 500.87,Z 269.207,A -85,B 0,C 180,E1 21462.124,E2 21462.124} C_VEL
LIN {X 0,Y 494.369,Z 256.682,A -85,B 0,C 180,E1 21460.635,E2 21460.635} C_VEL
LIN {X 0,Y 485.36,Z 236.103,A -85,B 0,C 180,E1 21458.171,E2 21458.171} C_VEL
LIN {X 0,Y 478.102,Z 221.559,A -85,B 0,C 180,E1 21456.139,E2 21456.139} C_VEL
LIN {X 0,Y 472.88,Z 212.154,A -85,B 0,C 180,E1 21454.644,E2 21454.644} C_VEL
LIN {X 0,Y 471.552,Z 212.636,A -85,B 0,C 180,E1 21454.481,E2 21454.481} C_VEL
LIN {X 0,Y 468.366,Z 214.69,A -85,B 0,C 180,E1 21454.156,E2 21454.156} C_VEL
LIN {X 0,Y 466.144,Z 214.924,A -85,B 0,C 180,E1 21453.822,E2 21453.822} C_VEL
LIN {X 0,Y 465.893,Z 214.868,A -85,B 0,C 180,E1 21453.768,E2 21453.768} C_VEL
LIN {X 0,Y 466.402,Z 250.859,A -85,B 0,C 180,E1 21450.961,E2 21450.961} C_VEL
LIN {X 0,Y 466.482,Z 287.915,A -85,B 0,C 180,E1 21447.926,E2 21447.926} C_VEL
LIN {X 0,Y 466.153,Z 322.409,A -85,B 0,C 180,E1 21444.995,E2 21444.995} C_VEL
LIN {X 0,Y 465.959,Z 333.18,A -85,B 0,C 180,E1 21444.06,E2 21444.06} C_VEL
LIN {X 0,Y 464.837,Z 338.496,A -85,B 0,C 180,E1 21443.713,E2 21443.713} C_VEL
LIN {X 0,Y 462.617,Z 449.855,A -85,B 0,C 180,E1 21441.645,E2 21441.645} C_VEL
LIN {X 0,Y 462.226,Z 503.167,A -85,B 0,C 180,E1 21440.703,E2 21440.703} C_VEL
LIN {X 0,Y 462.158,Z 520.604,A -85,B 0,C 180,E1 21440.182,E2 21440.182} C_VEL
LIN {X 0,Y 461.895,Z 536.738,A -85,B 0,C 180,E1 21439.473,E2 21439.473} C_VEL
LIN {X 0,Y 461.467,Z 553.168,A -85,B 0,C 180,E1 21438.507,E2 21438.507} C_VEL
LIN {X 0,Y 460.948,Z 567.548,A -85,B 0,C 180,E1 21437.418,E2 21437.418} C_VEL
LIN {X 0,Y 460.299,Z 581.556,A -85,B 0,C 180,E1 21436.078,E2 21436.078} C_VEL
LIN {X 0,Y 459.653,Z 593.925,A -85,B 0,C 180,E1 21434.615,E2 21434.615} C_VEL
LIN {X 0,Y 459.006,Z 605.229,A -85,B 0,C 180,E1 21432.965,E2 21432.965} C_VEL
LIN {X 0,Y 458.418,Z 614.883,A -85,B 0,C 180,E1 21431.193,E2 21431.193} C_VEL
LIN {X 0,Y 457.935,Z 623.113,A -85,B 0,C 180,E1 21429.282,E2 21429.282} C_VEL
LIN {X 0,Y 457.553,Z 629.706,A -85,B 0,C 180,E1 21427.281,E2 21427.281} C_VEL
LIN {X 0,Y 457.273,Z 634.433,A -85,B 0,C 180,E1 21425.269,E2 21425.269} C_VEL
LIN {X 0,Y 457.086,Z 637.627,A -85,B 0,C 180,E1 21423.134,E2 21423.134} C_VEL
LIN {X 0,Y 456.986,Z 639.077,A -85,B 0,C 180,E1 21421.003,E2 21421.003} C_VEL
LIN {X 0,Y 456.941,Z 638.786,A -85,B 0,C 180,E1 21418.871,E2 21418.871} C_VEL
LIN {X 0,Y 456.954,Z 636.664,A -85,B 0,C 180,E1 21416.664,E2 21416.664} C_VEL
LIN {X 0,Y 457.058,Z 632.74,A -85,B 0,C 180,E1 21414.476,E2 21414.476} C_VEL
LIN {X 0,Y 457.255,Z 627.367,A -85,B 0,C 180,E1 21412.461,E2 21412.461} C_VEL
LIN {X 0,Y 457.575,Z 620.108,A -85,B 0,C 180,E1 21410.44,E2 21410.44} C_VEL
LIN {X 0,Y 458.007,Z 611.369,A -85,B 0,C 180,E1 21408.541,E2 21408.541} C_VEL
LIN {X 0,Y 458.566,Z 601.171,A -85,B 0,C 180,E1 21406.765,E2 21406.765} C_VEL
LIN {X 0,Y 459.219,Z 589.414,A -85,B 0,C 180,E1 21405.112,E2 21405.112} C_VEL
LIN {X 0,Y 459.939,Z 576.07,A -85,B 0,C 180,E1 21403.584,E2 21403.584} C_VEL
LIN {X 0,Y 460.661,Z 561.659,A -85,B 0,C 180,E1 21402.244,E2 21402.244} C_VEL
LIN {X 0,Y 461.338,Z 545.837,A -85,B 0,C 180,E1 21401.079,E2 21401.079} C_VEL
LIN {X 0,Y 461.896,Z 529.326,A -85,B 0,C 180,E1 21400.131,E2 21400.131} C_VEL
LIN {X 0,Y 462.338,Z 512.011,A -85,B 0,C 180,E1 21399.396,E2 21399.396} C_VEL
LIN {X 0,Y 462.569,Z 493.98,A -85,B 0,C 180,E1 21398.884,E2 21398.884} C_VEL
LIN {X 0,Y 464.769,Z 330.794,A -85,B 0,C 180,E1 21396.055,E2 21396.055} C_VEL
LIN {X 0,Y 463.939,Z 325.437,A -85,B 0,C 180,E1 21395.895,E2 21395.895} C_VEL
LIN {X 0,Y 465.027,Z 288.217,A -85,B 0,C 180,E1 21392.357,E2 21392.357} C_VEL
LIN {X 0,Y 465.941,Z 255.401,A -85,B 0,C 180,E1 21389.234,E2 21389.234} C_VEL
LIN {X 0,Y 467.368,Z 256.898,A -85,B 0,C 180,E1 21389.035,E2 21389.035} C_VEL
LIN {X 0,Y 469.633,Z 256.897,A -85,B 0,C 180,E1 21388.773,E2 21388.773} C_VEL
LIN {X 0,Y 473.073,Z 254.691,A -85,B 0,C 180,E1 21388.43,E2 21388.43} C_VEL
LIN {X 0,Y 474.588,Z 253.413,A -85,B 0,C 180,E1 21388.288,E2 21388.288} C_VEL
LIN {X 0,Y 478.515,Z 252.92,A -85,B 0,C 180,E1 21387.874,E2 21387.874} C_VEL
LIN {X 0,Y 482.822,Z 250.424,A -85,B 0,C 180,E1 21387.47,E2 21387.47} C_VEL
LIN {X 0,Y 483.639,Z 250.177,A -85,B 0,C 180,E1 21387.39,E2 21387.39} C_VEL
LIN {X 0,Y 480.936,Z 351.773,A -85,B 0,C 180,E1 21385.612,E2 21385.612} C_VEL
LIN {X 0,Y 479.955,Z 359.457,A -85,B 0,C 180,E1 21385.55,E2 21385.55} C_VEL
LIN {X 0,Y 474.4,Z 379.958,A -85,B 0,C 180,E1 21385.649,E2 21385.649} C_VEL
LIN {X 0,Y 473.614,Z 386.554,A -85,B 0,C 180,E1 21385.587,E2 21385.587} C_VEL
LIN {X 0,Y 471.139,Z 475.079,A -85,B 0,C 180,E1 21383.979,E2 21383.979} C_VEL
LIN {X 0,Y 470.089,Z 496.438,A -85,B 0,C 180,E1 21383.358,E2 21383.358} C_VEL
LIN {X 0,Y 468.669,Z 517.345,A -85,B 0,C 180,E1 21382.526,E2 21382.526} C_VEL
LIN {X 0,Y 466.928,Z 537.359,A -85,B 0,C 180,E1 21381.506,E2 21381.506} C_VEL
LIN {X 0,Y 464.88,Z 557.041,A -85,B 0,C 180,E1 21380.256,E2 21380.256} C_VEL
LIN {X 0,Y 462.716,Z 575.107,A -85,B 0,C 180,E1 21378.856,E2 21378.856} C_VEL
LIN {X 0,Y 460.297,Z 593.482,A -85,B 0,C 180,E1 21377.164,E2 21377.164} C_VEL
LIN {X 0,Y 458.002,Z 610.246,A -85,B 0,C 180,E1 21375.335,E2 21375.335} C_VEL
LIN {X 0,Y 455.804,Z 625.57,A -85,B 0,C 180,E1 21373.362,E2 21373.362} C_VEL
LIN {X 0,Y 453.672,Z 640.859,A -85,B 0,C 180,E1 21371.054,E2 21371.054} C_VEL
LIN {X 0,Y 451.946,Z 653.647,A -85,B 0,C 180,E1 21368.763,E2 21368.763} C_VEL
LIN {X 0,Y 450.612,Z 664.56,A -85,B 0,C 180,E1 21366.489,E2 21366.489} C_VEL
LIN {X 0,Y 449.451,Z 676.091,A -85,B 0,C 180,E1 21363.693,E2 21363.693} C_VEL
LIN {X 0,Y 448.805,Z 683.985,A -85,B 0,C 180,E1 21361.421,E2 21361.421} C_VEL
LIN {X 0,Y 448.336,Z 691.636,A -85,B 0,C 180,E1 21358.782,E2 21358.782} C_VEL
LIN {X 0,Y 448.064,Z 697.624,A -85,B 0,C 180,E1 21356.079,E2 21356.079} C_VEL
LIN {X 0,Y 447.959,Z 701.647,A -85,B 0,C 180,E1 21353.689,E2 21353.689} C_VEL
LIN {X 0,Y 447.919,Z 704.718,A -85,B 0,C 180,E1 21351.063,E2 21351.063} C_VEL
LIN {X 0,Y 447.902,Z 706.225,A -85,B 0,C 180,E1 21348.346,E2 21348.346} C_VEL
LIN {X 0,Y 447.914,Z 706.331,A -85,B 0,C 180,E1 21346.07,E2 21346.07} C_VEL
LIN {X 0,Y 447.917,Z 705.305,A -85,B 0,C 180,E1 21343.687,E2 21343.687} C_VEL
LIN {X 0,Y 447.941,Z 702.502,A -85,B 0,C 180,E1 21340.807,E2 21340.807} C_VEL
LIN {X 0,Y 448.032,Z 698.344,A -85,B 0,C 180,E1 21338.212,E2 21338.212} C_VEL
LIN {X 0,Y 448.246,Z 693.25,A -85,B 0,C 180,E1 21335.812,E2 21335.812} C_VEL
LIN {X 0,Y 448.717,Z 685.427,A -85,B 0,C 180,E1 21332.938,E2 21332.938} C_VEL
LIN {X 0,Y 449.355,Z 677.178,A -85,B 0,C 180,E1 21330.51,E2 21330.51} C_VEL
LIN {X 0,Y 450.285,Z 667.489,A -85,B 0,C 180,E1 21328.091,E2 21328.091} C_VEL
LIN {X 0,Y 451.675,Z 655.729,A -85,B 0,C 180,E1 21325.557,E2 21325.557} C_VEL
LIN {X 0,Y 453.298,Z 643.38,A -85,B 0,C 180,E1 21323.287,E2 21323.287} C_VEL
LIN {X 0,Y 455.452,Z 628.098,A -85,B 0,C 180,E1 21320.906,E2 21320.906} C_VEL
LIN {X 0,Y 457.584,Z 612.983,A -85,B 0,C 180,E1 21318.914,E2 21318.914} C_VEL
LIN {X 0,Y 460.129,Z 594.772,A -85,B 0,C 180,E1 21316.875,E2 21316.875} C_VEL
LIN {X 0,Y 462.501,Z 577.237,A -85,B 0,C 180,E1 21315.221,E2 21315.221} C_VEL
LIN {X 0,Y 464.763,Z 558.729,A -85,B 0,C 180,E1 21313.759,E2 21313.759} C_VEL
LIN {X 0,Y 466.757,Z 540.232,A -85,B 0,C 180,E1 21312.549,E2 21312.549} C_VEL
LIN {X 0,Y 468.61,Z 520.668,A -85,B 0,C 180,E1 21311.495,E2 21311.495} C_VEL
LIN {X 0,Y 470.116,Z 500.985,A -85,B 0,C 180,E1 21310.663,E2 21310.663} C_VEL
LIN {X 0,Y 471.258,Z 480.036,A -85,B 0,C 180,E1 21309.998,E2 21309.998} C_VEL
LIN {X 0,Y 472.074,Z 457.614,A -85,B 0,C 180,E1 21309.511,E2 21309.511} C_VEL
LIN {X 0,Y 478.235,Z 249.726,A -85,B 0,C 180,E1 21305.793,E2 21305.793} C_VEL
LIN {X 0,Y 478.691,Z 230.15,A -85,B 0,C 180,E1 21305.433,E2 21305.433} C_VEL
LIN {X 0,Y 465.47,Z 210.226,A -85,B 0,C 180,E1 21303.536,E2 21303.536} C_VEL
LIN {X 0,Y 458.485,Z 200.727,A -85,B 0,C 180,E1 21302.504,E2 21302.504} C_VEL
LIN {X 0,Y 453.802,Z 195.058,A -85,B 0,C 180,E1 21301.803,E2 21301.803} C_VEL
LIN {X 0,Y 451.841,Z 191.386,A -85,B 0,C 180,E1 21301.013,E2 21301.013} C_VEL
LIN {X 0,Y 449.367,Z 187,A -85,B 0,C 180,E1 21300.024,E2 21300.024} C_VEL
LIN {X 0,Y 449.108,Z 185.792,A -85,B 0,C 180,E1 21299.792,E2 21299.792} C_VEL
LIN {X 0,Y 449.091,Z 185.791,A -85,B 0,C 180,E1 21296.146,E2 21296.146} C_VEL
LIN {X 0,Y 449.097,Z 185.782,A -85,B 0,C 180,E1 21292.409,E2 21292.409} C_VEL
LIN {X 0,Y 449.136,Z 185.775,A -85,B 0,C 180,E1 21288.78,E2 21288.78} C_VEL
LIN {X 0,Y 449.133,Z 185.775,A -85,B 0,C 180,E1 21285.068,E2 21285.068} C_VEL
LIN {X 0,Y 449.114,Z 185.78,A -85,B 0,C 180,E1 21281.387,E2 21281.387} C_VEL
LIN {X 0,Y 449.096,Z 185.787,A -85,B 0,C 180,E1 21277.592,E2 21277.592} C_VEL
LIN {X 0,Y 449.074,Z 185.795,A -85,B 0,C 180,E1 21273.823,E2 21273.823} C_VEL
LIN {X 0,Y 449.097,Z 185.793,A -85,B 0,C 180,E1 21270.062,E2 21270.062} C_VEL
LIN {X 0,Y 449.127,Z 185.782,A -85,B 0,C 180,E1 21266.44,E2 21266.44} C_VEL
LIN {X 0,Y 449.138,Z 185.768,A -85,B 0,C 180,E1 21262.652,E2 21262.652} C_VEL
LIN {X 0,Y 449.119,Z 185.78,A -85,B 0,C 180,E1 21258.886,E2 21258.886} C_VEL
LIN {X 0,Y 449.087,Z 185.794,A -85,B 0,C 180,E1 21255.232,E2 21255.232} C_VEL
LIN {X 0,Y 449.077,Z 185.794,A -85,B 0,C 180,E1 21251.56,E2 21251.56} C_VEL
LIN {X 0,Y 449.099,Z 185.783,A -85,B 0,C 180,E1 21247.806,E2 21247.806} C_VEL
LIN {X 0,Y 449.123,Z 185.772,A -85,B 0,C 180,E1 21244.086,E2 21244.086} C_VEL
LIN {X 0,Y 449.138,Z 185.776,A -85,B 0,C 180,E1 21240.383,E2 21240.383} C_VEL
LIN {X 0,Y 449.117,Z 185.784,A -85,B 0,C 180,E1 21236.682,E2 21236.682} C_VEL
LIN {X 0,Y 449.078,Z 185.794,A -85,B 0,C 180,E1 21233.095,E2 21233.095} C_VEL
LIN {X 0,Y 449.088,Z 185.795,A -85,B 0,C 180,E1 21229.481,E2 21229.481} C_VEL
LIN {X 0,Y 449.112,Z 185.787,A -85,B 0,C 180,E1 21225.693,E2 21225.693} C_VEL
LIN {X 0,Y 449.128,Z 185.779,A -85,B 0,C 180,E1 21221.915,E2 21221.915} C_VEL
LIN {X 0,Y 449.153,Z 185.91,A -85,B 0,C 180,E1 21218.382,E2 21218.382} C_VEL
LIN {X 0,Y 450.284,Z 189.022,A -85,B 0,C 180,E1 21217.812,E2 21217.812} C_VEL
LIN {X 0,Y 451.665,Z 190.971,A -85,B 0,C 180,E1 21217.345,E2 21217.345} C_VEL
LIN {X 0,Y 453.465,Z 194.638,A -85,B 0,C 180,E1 21216.617,E2 21216.617} C_VEL
LIN {X 0,Y 458.895,Z 205.038,A -85,B 0,C 180,E1 21214.582,E2 21214.582} C_VEL
LIN {X 0,Y 466.794,Z 220.859,A -85,B 0,C 180,E1 21211.747,E2 21211.747} C_VEL
LIN {X 0,Y 475.864,Z 240.45,A -85,B 0,C 180,E1 21208.595,E2 21208.595} C_VEL
LIN {X 0,Y 478.42,Z 246.268,A -85,B 0,C 180,E1 21207.726,E2 21207.726} C_VEL
LIN {X 0,Y 474.807,Z 287.766,A -85,B 0,C 180,E1 21204.242,E2 21204.242} C_VEL
LIN {X 0,Y 473.777,Z 309.014,A -85,B 0,C 180,E1 21202.418,E2 21202.418} C_VEL
LIN {X 0,Y 474.797,Z 326.522,A -85,B 0,C 180,E1 21200.75,E2 21200.75} C_VEL
LIN {X 0,Y 477.663,Z 341.732,A -85,B 0,C 180,E1 21199.146,E2 21199.146} C_VEL
LIN {X 0,Y 482.197,Z 355.291,A -85,B 0,C 180,E1 21197.577,E2 21197.577} C_VEL
LIN {X 0,Y 488.353,Z 367.274,A -85,B 0,C 180,E1 21196.047,E2 21196.047} C_VEL
LIN {X 0,Y 496.562,Z 378.237,A -85,B 0,C 180,E1 21194.485,E2 21194.485} C_VEL
LIN {X 0,Y 505.434,Z 386.813,A -85,B 0,C 180,E1 21193.117,E2 21193.117} C_VEL
LIN {X 0,Y 516.073,Z 394.341,A -85,B 0,C 180,E1 21191.763,E2 21191.763} C_VEL
LIN {X 0,Y 520.908,Z 397.229,A -85,B 0,C 180,E1 21191.212,E2 21191.212} C_VEL
LIN {X 0,Y 507.237,Z 416.204,A -85,B 0,C 180,E1 21190.727,E2 21190.727} C_VEL
LIN {X 0,Y 497.95,Z 431.412,A -85,B 0,C 180,E1 21190.207,E2 21190.207} C_VEL
LIN {X 0,Y 492.707,Z 441.237,A -85,B 0,C 180,E1 21189.81,E2 21189.81} C_VEL
LIN {X 0,Y 484.734,Z 454.942,A -85,B 0,C 180,E1 21189.29,E2 21189.29} C_VEL
LIN {X 0,Y 478.62,Z 468.332,A -85,B 0,C 180,E1 21188.655,E2 21188.655} C_VEL
LIN {X 0,Y 475.485,Z 475.753,A -85,B 0,C 180,E1 21188.317,E2 21188.317} C_VEL
LIN {X 0,Y 473.637,Z 495.073,A -85,B 0,C 180,E1 21188.127,E2 21188.127} C_VEL
LIN {X 0,Y 472.65,Z 523.57,A -85,B 0,C 180,E1 21187.592,E2 21187.592} C_VEL
LIN {X 0,Y 470.916,Z 547.611,A -85,B 0,C 180,E1 21186.942,E2 21186.942} C_VEL
LIN {X 0,Y 469.001,Z 570.161,A -85,B 0,C 180,E1 21186.101,E2 21186.101} C_VEL
LIN {X 0,Y 466.957,Z 591.394,A -85,B 0,C 180,E1 21185.094,E2 21185.094} C_VEL
LIN {X 0,Y 464.658,Z 613.377,A -85,B 0,C 180,E1 21183.804,E2 21183.804} C_VEL
LIN {X 0,Y 462.27,Z 634.597,A -85,B 0,C 180,E1 21182.293,E2 21182.293} C_VEL
LIN {X 0,Y 459.99,Z 654.091,A -85,B 0,C 180,E1 21180.638,E2 21180.638} C_VEL
LIN {X 0,Y 457.756,Z 672.581,A -85,B 0,C 180,E1 21178.792,E2 21178.792} C_VEL
LIN {X 0,Y 455.58,Z 690.609,A -85,B 0,C 180,E1 21176.675,E2 21176.675} C_VEL
LIN {X 0,Y 453.575,Z 707.378,A -85,B 0,C 180,E1 21174.344,E2 21174.344} C_VEL
LIN {X 0,Y 451.969,Z 721.501,A -85,B 0,C 180,E1 21172.041,E2 21172.041} C_VEL
LIN {X 0,Y 450.686,Z 733.725,A -85,B 0,C 180,E1 21169.707,E2 21169.707} C_VEL
LIN {X 0,Y 449.514,Z 745.408,A -85,B 0,C 180,E1 21166.941,E2 21166.941} C_VEL
LIN {X 0,Y 448.722,Z 755.353,A -85,B 0,C 180,E1 21164.056,E2 21164.056} C_VEL
LIN {X 0,Y 448.248,Z 763.213,A -85,B 0,C 180,E1 21161.19,E2 21161.19} C_VEL
LIN {X 0,Y 448.019,Z 769.389,A -85,B 0,C 180,E1 21158.211,E2 21158.211} C_VEL
LIN {X 0,Y 447.933,Z 773.439,A -85,B 0,C 180,E1 21155.379,E2 21155.379} C_VEL
LIN {X 0,Y 447.91,Z 775.715,A -85,B 0,C 180,E1 21152.687,E2 21152.687} C_VEL
LIN {X 0,Y 447.913,Z 776.5,A -85,B 0,C 180,E1 21150,E2 21150} C_VEL
LIN {X 0,Y 447.913,Z 775.646,A -85,B 0,C 180,E1 21147.185,E2 21147.185} C_VEL
LIN {X 0,Y 447.934,Z 773.286,A -85,B 0,C 180,E1 21144.492,E2 21144.492} C_VEL
LIN {X 0,Y 448.019,Z 769.388,A -85,B 0,C 180,E1 21141.788,E2 21141.788} C_VEL
LIN {X 0,Y 448.247,Z 763.213,A -85,B 0,C 180,E1 21138.81,E2 21138.81} C_VEL
LIN {X 0,Y 448.723,Z 755.353,A -85,B 0,C 180,E1 21135.943,E2 21135.943} C_VEL
LIN {X 0,Y 449.517,Z 745.408,A -85,B 0,C 180,E1 21133.059,E2 21133.059} C_VEL
LIN {X 0,Y 450.687,Z 733.724,A -85,B 0,C 180,E1 21130.292,E2 21130.292} C_VEL
LIN {X 0,Y 451.96,Z 721.46,A -85,B 0,C 180,E1 21127.962,E2 21127.962} C_VEL
LIN {X 0,Y 453.556,Z 707.148,A -85,B 0,C 180,E1 21125.654,E2 21125.654} C_VEL
LIN {X 0,Y 455.398,Z 691.204,A -85,B 0,C 180,E1 21123.461,E2 21123.461} C_VEL
LIN {X 0,Y 457.338,Z 674.615,A -85,B 0,C 180,E1 21121.506,E2 21121.506} C_VEL
LIN {X 0,Y 459.446,Z 656.334,A -85,B 0,C 180,E1 21119.676,E2 21119.676} C_VEL
LIN {X 0,Y 461.61,Z 637.091,A -85,B 0,C 180,E1 21118.022,E2 21118.022} C_VEL
LIN {X 0,Y 463.823,Z 616.576,A -85,B 0,C 180,E1 21116.538,E2 21116.538} C_VEL
LIN {X 0,Y 466.126,Z 593.678,A -85,B 0,C 180,E1 21115.168,E2 21115.168} C_VEL
LIN {X 0,Y 468.25,Z 571.13,A -85,B 0,C 180,E1 21114.078,E2 21114.078} C_VEL
LIN {X 0,Y 470.168,Z 547.603,A -85,B 0,C 180,E1 21113.198,E2 21113.198} C_VEL
LIN {X 0,Y 471.96,Z 522.469,A -85,B 0,C 180,E1 21112.51,E2 21112.51} C_VEL
LIN {X 0,Y 472.911,Z 496.921,A -85,B 0,C 180,E1 21112.013,E2 21112.013} C_VEL
LIN {X 0,Y 474.228,Z 474.03,A -85,B 0,C 180,E1 21111.717,E2 21111.717} C_VEL
LIN {X 0,Y 474.791,Z 468.885,A -85,B 0,C 180,E1 21111.67,E2 21111.67} C_VEL
LIN {X 0,Y 481.613,Z 444.643,A -85,B 0,C 180,E1 21110.79,E2 21110.79} C_VEL
LIN {X 0,Y 487.437,Z 428.126,A -85,B 0,C 180,E1 21110.285,E2 21110.285} C_VEL
LIN {X 0,Y 493.104,Z 410.14,A -85,B 0,C 180,E1 21109.696,E2 21109.696} C_VEL
LIN {X 0,Y 501.967,Z 388.128,A -85,B 0,C 180,E1 21109.13,E2 21109.13} C_VEL
LIN {X 0,Y 515.282,Z 359.912,A -85,B 0,C 180,E1 21108.572,E2 21108.572} C_VEL
LIN {X 0,Y 521.4,Z 347.6,A -85,B 0,C 180,E1 21108.358,E2 21108.358} C_VEL
LIN {X 0,Y 527.264,Z 331.002,A -85,B 0,C 180,E1 21107.906,E2 21107.906} C_VEL
LIN {X 0,Y 536.196,Z 309.698,A -85,B 0,C 180,E1 21107.439,E2 21107.439} C_VEL
LIN {X 0,Y 524.767,Z 303.198,A -85,B 0,C 180,E1 21106.23,E2 21106.23} C_VEL
LIN {X 0,Y 508.973,Z 291.006,A -85,B 0,C 180,E1 21104.217,E2 21104.217} C_VEL
LIN {X 0,Y 500.067,Z 281.326,A -85,B 0,C 180,E1 21102.794,E2 21102.794} C_VEL
LIN {X 0,Y 493.47,Z 271.447,A -85,B 0,C 180,E1 21101.495,E2 21101.495} C_VEL
LIN {X 0,Y 479.324,Z 240.018,A -85,B 0,C 180,E1 21097.675,E2 21097.675} C_VEL
LIN {X 0,Y 471.425,Z 224.162,A -85,B 0,C 180,E1 21095.381,E2 21095.381} C_VEL
LIN {X 0,Y 469.378,Z 220.864,A -85,B 0,C 180,E1 21094.812,E2 21094.812} C_VEL
LIN {X 0,Y 465.346,Z 222.616,A -85,B 0,C 180,E1 21094.334,E2 21094.334} C_VEL
LIN {X 0,Y 462.45,Z 224.799,A -85,B 0,C 180,E1 21094.054,E2 21094.054} C_VEL
LIN {X 0,Y 460.365,Z 225.546,A -85,B 0,C 180,E1 21093.779,E2 21093.779} C_VEL
LIN {X 0,Y 459.23,Z 225.492,A -85,B 0,C 180,E1 21093.574,E2 21093.574} C_VEL
LIN {X 0,Y 459.524,Z 262.511,A -85,B 0,C 180,E1 21090.607,E2 21090.607} C_VEL
LIN {X 0,Y 459.453,Z 296.846,A -85,B 0,C 180,E1 21087.755,E2 21087.755} C_VEL
LIN {X 0,Y 458.949,Z 334.366,A -85,B 0,C 180,E1 21084.52,E2 21084.52} C_VEL
LIN {X 0,Y 457.605,Z 340.662,A -85,B 0,C 180,E1 21084.112,E2 21084.112} C_VEL
LIN {X 0,Y 455.207,Z 447.163,A -85,B 0,C 180,E1 21082.057,E2 21082.057} C_VEL
LIN {X 0,Y 454.683,Z 504.246,A -85,B 0,C 180,E1 21081.017,E2 21081.017} C_VEL
LIN {X 0,Y 454.627,Z 521.93,A -85,B 0,C 180,E1 21080.487,E2 21080.487} C_VEL
LIN {X 0,Y 454.338,Z 538.934,A -85,B 0,C 180,E1 21079.724,E2 21079.724} C_VEL
LIN {X 0,Y 453.892,Z 554.951,A -85,B 0,C 180,E1 21078.76,E2 21078.76} C_VEL
LIN {X 0,Y 453.357,Z 568.974,A -85,B 0,C 180,E1 21077.681,E2 21077.681} C_VEL
LIN {X 0,Y 452.694,Z 582.71,A -85,B 0,C 180,E1 21076.356,E2 21076.356} C_VEL
LIN {X 0,Y 451.99,Z 595.494,A -85,B 0,C 180,E1 21074.826,E2 21074.826} C_VEL
LIN {X 0,Y 451.314,Z 606.551,A -85,B 0,C 180,E1 21073.19,E2 21073.19} C_VEL
LIN {X 0,Y 450.679,Z 616.244,A -85,B 0,C 180,E1 21071.388,E2 21071.388} C_VEL
LIN {X 0,Y 450.159,Z 624.453,A -85,B 0,C 180,E1 21069.46,E2 21069.46} C_VEL
LIN {X 0,Y 449.74,Z 631.132,A -85,B 0,C 180,E1 21067.408,E2 21067.408} C_VEL
LIN {X 0,Y 449.43,Z 635.853,A -85,B 0,C 180,E1 21065.361,E2 21065.361} C_VEL
LIN {X 0,Y 449.22,Z 639.026,A -85,B 0,C 180,E1 21063.189,E2 21063.189} C_VEL
LIN {X 0,Y 449.105,Z 640.447,A -85,B 0,C 180,E1 21061.02,E2 21061.02} C_VEL
LIN {X 0,Y 449.053,Z 640.116,A -85,B 0,C 180,E1 21058.851,E2 21058.851} C_VEL
LIN {X 0,Y 449.065,Z 638.009,A -85,B 0,C 180,E1 21056.66,E2 21056.66} C_VEL
LIN {X 0,Y 449.167,Z 634.213,A -85,B 0,C 180,E1 21054.507,E2 21054.507} C_VEL
LIN {X 0,Y 449.375,Z 628.893,A -85,B 0,C 180,E1 21052.456,E2 21052.456} C_VEL
LIN {X 0,Y 449.711,Z 621.658,A -85,B 0,C 180,E1 21050.401,E2 21050.401} C_VEL
LIN {X 0,Y 450.192,Z 612.413,A -85,B 0,C 180,E1 21048.364,E2 21048.364} C_VEL
LIN {X 0,Y 450.793,Z 601.956,A -85,B 0,C 180,E1 21046.532,E2 21046.532} C_VEL
LIN {X 0,Y 451.486,Z 590.055,A -85,B 0,C 180,E1 21044.851,E2 21044.851} C_VEL
LIN {X 0,Y 452.25,Z 576.553,A -85,B 0,C 180,E1 21043.297,E2 21043.297} C_VEL
LIN {X 0,Y 453.007,Z 561.893,A -85,B 0,C 180,E1 21041.934,E2 21041.934} C_VEL
LIN {X 0,Y 453.704,Z 546.255,A -85,B 0,C 180,E1 21040.778,E2 21040.778} C_VEL
LIN {X 0,Y 454.275,Z 530.018,A -85,B 0,C 180,E1 21039.84,E2 21039.84} C_VEL
LIN {X 0,Y 454.725,Z 512.771,A -85,B 0,C 180,E1 21039.102,E2 21039.102} C_VEL
LIN {X 0,Y 454.965,Z 494.661,A -85,B 0,C 180,E1 21038.583,E2 21038.583} C_VEL
LIN {X 0,Y 457.321,Z 331.723,A -85,B 0,C 180,E1 21035.695,E2 21035.695} C_VEL
LIN {X 0,Y 456.512,Z 326.607,A -85,B 0,C 180,E1 21035.546,E2 21035.546} C_VEL
LIN {X 0,Y 457.64,Z 289.09,A -85,B 0,C 180,E1 21031.966,E2 21031.966} C_VEL
LIN {X 0,Y 458.34,Z 267.638,A -85,B 0,C 180,E1 21029.884,E2 21029.884} C_VEL
LIN {X 0,Y 459.998,Z 269.025,A -85,B 0,C 180,E1 21029.647,E2 21029.647} C_VEL
LIN {X 0,Y 462.657,Z 268.536,A -85,B 0,C 180,E1 21029.334,E2 21029.334} C_VEL
LIN {X 0,Y 466.368,Z 265.525,A -85,B 0,C 180,E1 21028.961,E2 21028.961} C_VEL
LIN {X 0,Y 467.198,Z 265.006,A -85,B 0,C 180,E1 21028.876,E2 21028.876} C_VEL
LIN {X 0,Y 471.051,Z 264.344,A -85,B 0,C 180,E1 21028.451,E2 21028.451} C_VEL
LIN {X 0,Y 475.385,Z 261.637,A -85,B 0,C 180,E1 21028.028,E2 21028.028} C_VEL
LIN {X 0,Y 477.311,Z 261.301,A -85,B 0,C 180,E1 21027.829,E2 21027.829} C_VEL
LIN {X 0,Y 473.614,Z 386.554,A -85,B 0,C 180,E1 21025.587,E2 21025.587} C_VEL
LIN {X 0,Y 472.603,Z 394.237,A -85,B 0,C 180,E1 21025.524,E2 21025.524} C_VEL
LIN {X 0,Y 467.011,Z 414.722,A -85,B 0,C 180,E1 21025.619,E2 21025.619} C_VEL
LIN {X 0,Y 466.209,Z 421.313,A -85,B 0,C 180,E1 21025.555,E2 21025.555} C_VEL
LIN {X 0,Y 464.484,Z 477.688,A -85,B 0,C 180,E1 21024.485,E2 21024.485} C_VEL
LIN {X 0,Y 463.398,Z 498.955,A -85,B 0,C 180,E1 21023.844,E2 21023.844} C_VEL
LIN {X 0,Y 461.902,Z 519.501,A -85,B 0,C 180,E1 21023.002,E2 21023.002} C_VEL
LIN {X 0,Y 460.021,Z 539.747,A -85,B 0,C 180,E1 21021.939,E2 21021.939} C_VEL
LIN {X 0,Y 457.96,Z 558.602,A -85,B 0,C 180,E1 21020.716,E2 21020.716} C_VEL
LIN {X 0,Y 455.69,Z 576.593,A -85,B 0,C 180,E1 21019.296,E2 21019.296} C_VEL
LIN {X 0,Y 453.137,Z 594.999,A -85,B 0,C 180,E1 21017.569,E2 21017.569} C_VEL
LIN {X 0,Y 450.653,Z 612.086,A -85,B 0,C 180,E1 21015.662,E2 21015.662} C_VEL
LIN {X 0,Y 448.345,Z 627.396,A -85,B 0,C 180,E1 21013.648,E2 21013.648} C_VEL
LIN {X 0,Y 446.118,Z 642.281,A -85,B 0,C 180,E1 21011.338,E2 21011.338} C_VEL
LIN {X 0,Y 444.217,Z 655.538,A -85,B 0,C 180,E1 21008.902,E2 21008.902} C_VEL
LIN {X 0,Y 442.646,Z 667.711,A -85,B 0,C 180,E1 21006.253,E2 21006.253} C_VEL
LIN {X 0,Y 441.553,Z 677.1,A -85,B 0,C 180,E1 21003.793,E2 21003.793} C_VEL
LIN {X 0,Y 440.709,Z 686.616,A -85,B 0,C 180,E1 21000.847,E2 21000.847} C_VEL
LIN {X 0,Y 440.26,Z 693.503,A -85,B 0,C 180,E1 20998.189,E2 20998.189} C_VEL
LIN {X 0,Y 440.052,Z 698.329,A -85,B 0,C 180,E1 20995.865,E2 20995.865} C_VEL
LIN {X 0,Y 439.946,Z 702.593,A -85,B 0,C 180,E1 20993.152,E2 20993.152} C_VEL
LIN {X 0,Y 439.914,Z 705.258,A -85,B 0,C 180,E1 20990.35,E2 20990.35} C_VEL
LIN {X 0,Y 439.907,Z 706.298,A -85,B 0,C 180,E1 20988.006,E2 20988.006} C_VEL
LIN {X 0,Y 439.906,Z 706.256,A -85,B 0,C 180,E1 20985.693,E2 20985.693} C_VEL
LIN {X 0,Y 439.914,Z 704.804,A -85,B 0,C 180,E1 20982.87,E2 20982.87} C_VEL
LIN {X 0,Y 439.956,Z 701.803,A -85,B 0,C 180,E1 20980.211,E2 20980.211} C_VEL
LIN {X 0,Y 440.068,Z 697.94,A -85,B 0,C 180,E1 20977.835,E2 20977.835} C_VEL
LIN {X 0,Y 440.339,Z 692.346,A -85,B 0,C 180,E1 20975.211,E2 20975.211} C_VEL
LIN {X 0,Y 440.831,Z 684.758,A -85,B 0,C 180,E1 20972.47,E2 20972.47} C_VEL
LIN {X 0,Y 441.682,Z 675.78,A -85,B 0,C 180,E1 20969.741,E2 20969.741} C_VEL
LIN {X 0,Y 442.959,Z 664.947,A -85,B 0,C 180,E1 20967.024,E2 20967.024} C_VEL
LIN {X 0,Y 444.422,Z 653.966,A -85,B 0,C 180,E1 20964.708,E2 20964.708} C_VEL
LIN {X 0,Y 446.375,Z 640.443,A -85,B 0,C 180,E1 20962.276,E2 20962.276} C_VEL
LIN {X 0,Y 448.622,Z 625.39,A -85,B 0,C 180,E1 20959.989,E2 20959.989} C_VEL
LIN {X 0,Y 451.077,Z 609.291,A -85,B 0,C 180,E1 20957.909,E2 20957.909} C_VEL
LIN {X 0,Y 453.504,Z 592.631,A -85,B 0,C 180,E1 20956.095,E2 20956.095} C_VEL
LIN {X 0,Y 455.925,Z 575.18,A -85,B 0,C 180,E1 20954.482,E2 20954.482} C_VEL
LIN {X 0,Y 458.238,Z 557.102,A -85,B 0,C 180,E1 20953.065,E2 20953.065} C_VEL
LIN {X 0,Y 460.365,Z 538.108,A -85,B 0,C 180,E1 20951.841,E2 20951.841} C_VEL
LIN {X 0,Y 462.243,Z 518.274,A -85,B 0,C 180,E1 20950.805,E2 20950.805} C_VEL
LIN {X 0,Y 463.792,Z 497.974,A -85,B 0,C 180,E1 20949.971,E2 20949.971} C_VEL
LIN {X 0,Y 464.936,Z 476.658,A -85,B 0,C 180,E1 20949.327,E2 20949.327} C_VEL
LIN {X 0,Y 466.125,Z 439.998,A -85,B 0,C 180,E1 20948.616,E2 20948.616} C_VEL
LIN {X 0,Y 472.31,Z 248.11,A -85,B 0,C 180,E1 20945.119,E2 20945.119} C_VEL
LIN {X 0,Y 472.628,Z 233.535,A -85,B 0,C 180,E1 20944.844,E2 20944.844} C_VEL
LIN {X 0,Y 457.829,Z 211.459,A -85,B 0,C 180,E1 20942.662,E2 20942.662} C_VEL
LIN {X 0,Y 453.285,Z 205.824,A -85,B 0,C 180,E1 20941.985,E2 20941.985} C_VEL
LIN {X 0,Y 448.985,Z 200.713,A -85,B 0,C 180,E1 20941.333,E2 20941.333} C_VEL
LIN {X 0,Y 446.824,Z 197.989,A -85,B 0,C 180,E1 20940.95,E2 20940.95} C_VEL
LIN {X 0,Y 445.757,Z 195.871,A -85,B 0,C 180,E1 20940.495,E2 20940.495} C_VEL
LIN {X 0,Y 443.364,Z 191.365,A -85,B 0,C 180,E1 20939.483,E2 20939.483} C_VEL
LIN {X 0,Y 441.586,Z 188.422,A -85,B 0,C 180,E1 20938.768,E2 20938.768} C_VEL
LIN {X 0,Y 441.19,Z 186.766,A -85,B 0,C 180,E1 20938.432,E2 20938.432} C_VEL
LIN {X 0,Y 441.172,Z 186.768,A -85,B 0,C 180,E1 20934.677,E2 20934.677} C_VEL
LIN {X 0,Y 441.197,Z 186.771,A -85,B 0,C 180,E1 20930.811,E2 20930.811} C_VEL
LIN {X 0,Y 441.198,Z 186.775,A -85,B 0,C 180,E1 20927.055,E2 20927.055} C_VEL
LIN {X 0,Y 441.188,Z 186.774,A -85,B 0,C 180,E1 20923.325,E2 20923.325} C_VEL
LIN {X 0,Y 441.168,Z 186.773,A -85,B 0,C 180,E1 20919.558,E2 20919.558} C_VEL
LIN {X 0,Y 441.144,Z 186.77,A -85,B 0,C 180,E1 20915.787,E2 20915.787} C_VEL
LIN {X 0,Y 441.144,Z 186.765,A -85,B 0,C 180,E1 20912.031,E2 20912.031} C_VEL
LIN {X 0,Y 441.181,Z 186.771,A -85,B 0,C 180,E1 20908.42,E2 20908.42} C_VEL
LIN {X 0,Y 441.197,Z 186.776,A -85,B 0,C 180,E1 20904.645,E2 20904.645} C_VEL
LIN {X 0,Y 441.184,Z 186.778,A -85,B 0,C 180,E1 20900.978,E2 20900.978} C_VEL
LIN {X 0,Y 441.158,Z 186.77,A -85,B 0,C 180,E1 20897.272,E2 20897.272} C_VEL
LIN {X 0,Y 441.131,Z 186.766,A -85,B 0,C 180,E1 20893.501,E2 20893.501} C_VEL
LIN {X 0,Y 441.151,Z 186.776,A -85,B 0,C 180,E1 20889.787,E2 20889.787} C_VEL
LIN {X 0,Y 441.175,Z 186.78,A -85,B 0,C 180,E1 20885.985,E2 20885.985} C_VEL
LIN {X 0,Y 441.194,Z 186.778,A -85,B 0,C 180,E1 20882.208,E2 20882.208} C_VEL
LIN {X 0,Y 441.196,Z 186.774,A -85,B 0,C 180,E1 20878.442,E2 20878.442} C_VEL
LIN {X 0,Y 441.173,Z 186.773,A -85,B 0,C 180,E1 20874.669,E2 20874.669} C_VEL
LIN {X 0,Y 441.151,Z 186.773,A -85,B 0,C 180,E1 20871.003,E2 20871.003} C_VEL
LIN {X 0,Y 441.171,Z 186.773,A -85,B 0,C 180,E1 20867.301,E2 20867.301} C_VEL
LIN {X 0,Y 441.187,Z 186.778,A -85,B 0,C 180,E1 20863.544,E2 20863.544} C_VEL
LIN {X 0,Y 441.196,Z 186.774,A -85,B 0,C 180,E1 20859.713,E2 20859.713} C_VEL
LIN {X 0,Y 442.353,Z 190.057,A -85,B 0,C 180,E1 20859.076,E2 20859.076} C_VEL
LIN {X 0,Y 443.794,Z 191.867,A -85,B 0,C 180,E1 20858.594,E2 20858.594} C_VEL
LIN {X 0,Y 445.493,Z 195.552,A -85,B 0,C 180,E1 20857.849,E2 20857.849} C_VEL
LIN {X 0,Y 446.715,Z 197.883,A -85,B 0,C 180,E1 20857.358,E2 20857.358} C_VEL
LIN {X 0,Y 449.215,Z 202.617,A -85,B 0,C 180,E1 20856.382,E2 20856.382} C_VEL
LIN {X 0,Y 455.644,Z 215.031,A -85,B 0,C 180,E1 20853.968,E2 20853.968} C_VEL
LIN {X 0,Y 464.178,Z 232.757,A -85,B 0,C 180,E1 20850.869,E2 20850.869} C_VEL
LIN {X 0,Y 472,Z 250.094,A -85,B 0,C 180,E1 20848.13,E2 20848.13} C_VEL
LIN {X 0,Y 468.237,Z 291.244,A -85,B 0,C 180,E1 20844.642,E2 20844.642} C_VEL
LIN {X 0,Y 467.176,Z 313.2,A -85,B 0,C 180,E1 20842.722,E2 20842.722} C_VEL
LIN {X 0,Y 468.287,Z 330.907,A -85,B 0,C 180,E1 20841.004,E2 20841.004} C_VEL
LIN {X 0,Y 471.246,Z 346.282,A -85,B 0,C 180,E1 20839.355,E2 20839.355} C_VEL
LIN {X 0,Y 475.847,Z 359.951,A -85,B 0,C 180,E1 20837.749,E2 20837.749} C_VEL
LIN {X 0,Y 482.148,Z 372.23,A -85,B 0,C 180,E1 20836.161,E2 20836.161} C_VEL
LIN {X 0,Y 490.157,Z 383.052,A -85,B 0,C 180,E1 20834.609,E2 20834.609} C_VEL
LIN {X 0,Y 499.167,Z 391.973,A -85,B 0,C 180,E1 20833.188,E2 20833.188} C_VEL
LIN {X 0,Y 510.42,Z 400.113,A -85,B 0,C 180,E1 20831.726,E2 20831.726} C_VEL
LIN {X 0,Y 510.927,Z 400.592,A -85,B 0,C 180,E1 20831.654,E2 20831.654} C_VEL
LIN {X 0,Y 498.836,Z 417.971,A -85,B 0,C 180,E1 20831.181,E2 20831.181} C_VEL
LIN {X 0,Y 489.877,Z 433.314,A -85,B 0,C 180,E1 20830.624,E2 20830.624} C_VEL
LIN {X 0,Y 486.311,Z 439.846,A -85,B 0,C 180,E1 20830.364,E2 20830.364} C_VEL
LIN {X 0,Y 477.923,Z 454.394,A -85,B 0,C 180,E1 20829.805,E2 20829.805} C_VEL
LIN {X 0,Y 469.623,Z 472.952,A -85,B 0,C 180,E1 20828.935,E2 20828.935} C_VEL
LIN {X 0,Y 467.537,Z 491.474,A -85,B 0,C 180,E1 20828.78,E2 20828.78} C_VEL
LIN {X 0,Y 466.408,Z 520.357,A -85,B 0,C 180,E1 20828.248,E2 20828.248} C_VEL
LIN {X 0,Y 464.602,Z 544.644,A -85,B 0,C 180,E1 20827.6,E2 20827.6} C_VEL
LIN {X 0,Y 462.489,Z 567.762,A -85,B 0,C 180,E1 20826.746,E2 20826.746} C_VEL
LIN {X 0,Y 460.223,Z 589.997,A -85,B 0,C 180,E1 20825.685,E2 20825.685} C_VEL
LIN {X 0,Y 457.733,Z 612.206,A -85,B 0,C 180,E1 20824.371,E2 20824.371} C_VEL
LIN {X 0,Y 455.331,Z 632.449,A -85,B 0,C 180,E1 20822.921,E2 20822.921} C_VEL
LIN {X 0,Y 452.885,Z 652.106,A -85,B 0,C 180,E1 20821.253,E2 20821.253} C_VEL
LIN {X 0,Y 450.498,Z 670.834,A -85,B 0,C 180,E1 20819.373,E2 20819.373} C_VEL
LIN {X 0,Y 448.149,Z 689.099,A -85,B 0,C 180,E1 20817.218,E2 20817.218} C_VEL
LIN {X 0,Y 445.928,Z 706.647,A -85,B 0,C 180,E1 20814.758,E2 20814.758} C_VEL
LIN {X 0,Y 444.094,Z 721.849,A -85,B 0,C 180,E1 20812.225,E2 20812.225} C_VEL
LIN {X 0,Y 442.732,Z 734.182,A -85,B 0,C 180,E1 20809.801,E2 20809.801} C_VEL
LIN {X 0,Y 441.621,Z 745.515,A -85,B 0,C 180,E1 20807.17,E2 20807.17} C_VEL
LIN {X 0,Y 440.892,Z 754.109,A -85,B 0,C 180,E1 20804.714,E2 20804.714} C_VEL
LIN {X 0,Y 440.355,Z 761.91,A -85,B 0,C 180,E1 20801.924,E2 20801.924} C_VEL
LIN {X 0,Y 440.073,Z 767.957,A -85,B 0,C 180,E1 20799.151,E2 20799.151} C_VEL
LIN {X 0,Y 439.945,Z 772.519,A -85,B 0,C 180,E1 20796.263,E2 20796.263} C_VEL
LIN {X 0,Y 439.913,Z 775.322,A -85,B 0,C 180,E1 20793.388,E2 20793.388} C_VEL
LIN {X 0,Y 439.9,Z 776.433,A -85,B 0,C 180,E1 20790.651,E2 20790.651} C_VEL
LIN {X 0,Y 439.909,Z 776.059,A -85,B 0,C 180,E1 20787.916,E2 20787.916} C_VEL
LIN {X 0,Y 439.928,Z 773.995,A -85,B 0,C 180,E1 20785.045,E2 20785.045} C_VEL
LIN {X 0,Y 439.993,Z 770.442,A -85,B 0,C 180,E1 20782.295,E2 20782.295} C_VEL
LIN {X 0,Y 440.184,Z 765.302,A -85,B 0,C 180,E1 20779.53,E2 20779.53} C_VEL
LIN {X 0,Y 440.602,Z 758.075,A -85,B 0,C 180,E1 20776.616,E2 20776.616} C_VEL
LIN {X 0,Y 441.303,Z 749.239,A -85,B 0,C 180,E1 20773.818,E2 20773.818} C_VEL
LIN {X 0,Y 442.231,Z 739.006,A -85,B 0,C 180,E1 20771.273,E2 20771.273} C_VEL
LIN {X 0,Y 443.506,Z 726.721,A -85,B 0,C 180,E1 20768.717,E2 20768.717} C_VEL
LIN {X 0,Y 445.08,Z 712.901,A -85,B 0,C 180,E1 20766.289,E2 20766.289} C_VEL
LIN {X 0,Y 446.935,Z 697.532,A -85,B 0,C 180,E1 20763.993,E2 20763.993} C_VEL
LIN {X 0,Y 449.034,Z 680.551,A -85,B 0,C 180,E1 20761.832,E2 20761.832} C_VEL
LIN {X 0,Y 451.39,Z 661.289,A -85,B 0,C 180,E1 20759.754,E2 20759.754} C_VEL
LIN {X 0,Y 453.721,Z 642.025,A -85,B 0,C 180,E1 20758.003,E2 20758.003} C_VEL
LIN {X 0,Y 456.158,Z 620.809,A -85,B 0,C 180,E1 20756.37,E2 20756.37} C_VEL
LIN {X 0,Y 458.511,Z 599.386,A -85,B 0,C 180,E1 20755.004,E2 20755.004} C_VEL
LIN {X 0,Y 460.816,Z 576.667,A -85,B 0,C 180,E1 20753.818,E2 20753.818} C_VEL
LIN {X 0,Y 462.994,Z 553.685,A -85,B 0,C 180,E1 20752.864,E2 20752.864} C_VEL
LIN {X 0,Y 464.907,Z 529.862,A -85,B 0,C 180,E1 20752.128,E2 20752.128} C_VEL
LIN {X 0,Y 466.329,Z 503.823,A -85,B 0,C 180,E1 20751.545,E2 20751.545} C_VEL
LIN {X 0,Y 467.188,Z 484.017,A -85,B 0,C 180,E1 20751.237,E2 20751.237} C_VEL
LIN {X 0,Y 468.934,Z 465.22,A -85,B 0,C 180,E1 20751.043,E2 20751.043} C_VEL
LIN {X 0,Y 474.837,Z 444.296,A -85,B 0,C 180,E1 20750.277,E2 20750.277} C_VEL
LIN {X 0,Y 481.047,Z 426.559,A -85,B 0,C 180,E1 20749.728,E2 20749.728} C_VEL
LIN {X 0,Y 486.82,Z 408.613,A -85,B 0,C 180,E1 20749.144,E2 20749.144} C_VEL
LIN {X 0,Y 495.736,Z 386.591,A -85,B 0,C 180,E1 20748.581,E2 20748.581} C_VEL
LIN {X 0,Y 509.086,Z 358.33,A -85,B 0,C 180,E1 20748.029,E2 20748.029} C_VEL
LIN {X 0,Y 515.197,Z 346.018,A -85,B 0,C 180,E1 20747.817,E2 20747.817} C_VEL
LIN {X 0,Y 521.606,Z 328.281,A -85,B 0,C 180,E1 20747.342,E2 20747.342} C_VEL
LIN {X 0,Y 527.47,Z 314.176,A -85,B 0,C 180,E1 20747.028,E2 20747.028} C_VEL
LIN {X 0,Y 516.337,Z 307.016,A -85,B 0,C 180,E1 20745.765,E2 20745.765} C_VEL
LIN {X 0,Y 502.78,Z 296.097,A -85,B 0,C 180,E1 20743.95,E2 20743.95} C_VEL
LIN {X 0,Y 493.62,Z 285.642,A -85,B 0,C 180,E1 20742.416,E2 20742.416} C_VEL
LIN {X 0,Y 487.123,Z 275.314,A -85,B 0,C 180,E1 20741.058,E2 20741.058} C_VEL
LIN {X 0,Y 474.503,Z 246.505,A -85,B 0,C 180,E1 20737.515,E2 20737.515} C_VEL
LIN {X 0,Y 467.464,Z 232.08,A -85,B 0,C 180,E1 20735.42,E2 20735.42} C_VEL
LIN {X 0,Y 465.778,Z 229.159,A -85,B 0,C 180,E1 20734.932,E2 20734.932} C_VEL
LIN {X 0,Y 461.188,Z 232.082,A -85,B 0,C 180,E1 20734.461,E2 20734.461} C_VEL
LIN {X 0,Y 459.105,Z 232.777,A -85,B 0,C 180,E1 20734.186,E2 20734.186} C_VEL
LIN {X 0,Y 455.789,Z 235.321,A -85,B 0,C 180,E1 20733.862,E2 20733.862} C_VEL
LIN {X 0,Y 453.454,Z 236.093,A -85,B 0,C 180,E1 20733.541,E2 20733.541} C_VEL
LIN {X 0,Y 452.639,Z 236.083,A -85,B 0,C 180,E1 20733.385,E2 20733.385} C_VEL
LIN {X 0,Y 452.686,Z 275.444,A -85,B 0,C 180,E1 20730.164,E2 20730.164} C_VEL
LIN {X 0,Y 452.336,Z 313.33,A -85,B 0,C 180,E1 20726.945,E2 20726.945} C_VEL
LIN {X 0,Y 451.787,Z 336.512,A -85,B 0,C 180,E1 20724.935,E2 20724.935} C_VEL
LIN {X 0,Y 450.422,Z 342.792,A -85,B 0,C 180,E1 20724.53,E2 20724.53} C_VEL
LIN {X 0,Y 447.795,Z 447.435,A -85,B 0,C 180,E1 20722.437,E2 20722.437} C_VEL
LIN {X 0,Y 447.18,Z 505.265,A -85,B 0,C 180,E1 20721.352,E2 20721.352} C_VEL
LIN {X 0,Y 447.123,Z 523.291,A -85,B 0,C 180,E1 20720.806,E2 20720.806} C_VEL
LIN {X 0,Y 446.84,Z 539.602,A -85,B 0,C 180,E1 20720.07,E2 20720.07} C_VEL
LIN {X 0,Y 446.37,Z 555.846,A -85,B 0,C 180,E1 20719.089,E2 20719.089} C_VEL
LIN {X 0,Y 445.799,Z 570.409,A -85,B 0,C 180,E1 20717.962,E2 20717.962} C_VEL
LIN {X 0,Y 445.103,Z 584.052,A -85,B 0,C 180,E1 20716.629,E2 20716.629} C_VEL
LIN {X 0,Y 444.344,Z 596.945,A -85,B 0,C 180,E1 20715.064,E2 20715.064} C_VEL
LIN {X 0,Y 443.636,Z 607.908,A -85,B 0,C 180,E1 20713.423,E2 20713.423} C_VEL
LIN {X 0,Y 442.953,Z 617.713,A -85,B 0,C 180,E1 20711.577,E2 20711.577} C_VEL
LIN {X 0,Y 442.388,Z 625.876,A -85,B 0,C 180,E1 20709.628,E2 20709.628} C_VEL
LIN {X 0,Y 441.929,Z 632.557,A -85,B 0,C 180,E1 20707.54,E2 20707.54} C_VEL
LIN {X 0,Y 441.589,Z 637.284,A -85,B 0,C 180,E1 20705.457,E2 20705.457} C_VEL
LIN {X 0,Y 441.357,Z 640.443,A -85,B 0,C 180,E1 20703.246,E2 20703.246} C_VEL
LIN {X 0,Y 441.227,Z 641.833,A -85,B 0,C 180,E1 20701.038,E2 20701.038} C_VEL
LIN {X 0,Y 441.166,Z 641.446,A -85,B 0,C 180,E1 20698.831,E2 20698.831} C_VEL
LIN {X 0,Y 441.177,Z 639.31,A -85,B 0,C 180,E1 20696.621,E2 20696.621} C_VEL
LIN {X 0,Y 441.288,Z 635.419,A -85,B 0,C 180,E1 20694.408,E2 20694.408} C_VEL
LIN {X 0,Y 441.51,Z 630.005,A -85,B 0,C 180,E1 20692.321,E2 20692.321} C_VEL
LIN {X 0,Y 441.868,Z 622.664,A -85,B 0,C 180,E1 20690.229,E2 20690.229} C_VEL
LIN {X 0,Y 442.353,Z 613.84,A -85,B 0,C 180,E1 20688.262,E2 20688.262} C_VEL
LIN {X 0,Y 442.974,Z 603.546,A -85,B 0,C 180,E1 20686.423,E2 20686.423} C_VEL
LIN {X 0,Y 443.71,Z 591.415,A -85,B 0,C 180,E1 20684.68,E2 20684.68} C_VEL
LIN {X 0,Y 444.527,Z 577.582,A -85,B 0,C 180,E1 20683.065,E2 20683.065} C_VEL
